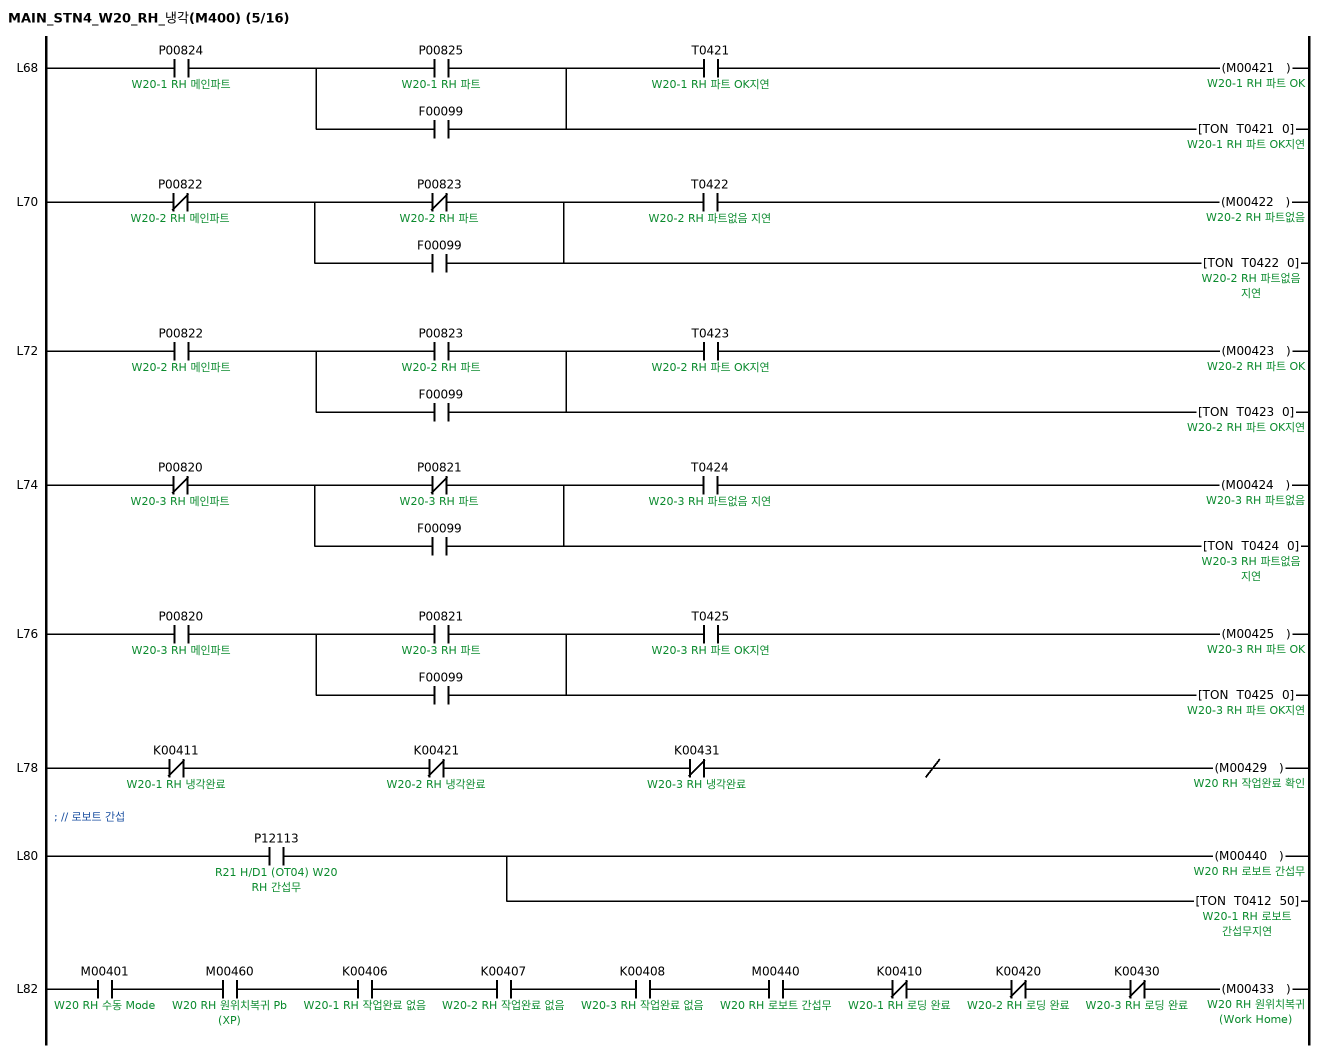
[picture p96: MAIN_STN4_W20_RH_냉각(M400) rungs L68-L82]
; L68
LOAD      P00824	// W20-1 RH 메인파트
LOAD      P00825	// W20-1 RH 파트
OR        F00099
AND LOAD
MPUSH
AND       T0421	// W20-1 RH 파트 OK지연
OUT       M00421	// W20-1 RH 파트 OK
MPOP
TON       T0421 0	// W20-1 RH 파트 OK지연
; L70
LOAD NOT  P00822	// W20-2 RH 메인파트
LOAD NOT  P00823	// W20-2 RH 파트
OR        F00099
AND LOAD
MPUSH
AND       T0422	// W20-2 RH 파트없음 지연
OUT       M00422	// W20-2 RH 파트없음
MPOP
TON       T0422 0	// W20-2 RH 파트없음 지연
; L72
LOAD      P00822	// W20-2 RH 메인파트
LOAD      P00823	// W20-2 RH 파트
OR        F00099
AND LOAD
MPUSH
AND       T0423	// W20-2 RH 파트 OK지연
OUT       M00423	// W20-2 RH 파트 OK
MPOP
TON       T0423 0	// W20-2 RH 파트 OK지연
; L74
LOAD NOT  P00820	// W20-3 RH 메인파트
LOAD NOT  P00821	// W20-3 RH 파트
OR        F00099
AND LOAD
MPUSH
AND       T0424	// W20-3 RH 파트없음 지연
OUT       M00424	// W20-3 RH 파트없음
MPOP
TON       T0424 0	// W20-3 RH 파트없음 지연
; L76
LOAD      P00820	// W20-3 RH 메인파트
LOAD      P00821	// W20-3 RH 파트
OR        F00099
AND LOAD
MPUSH
AND       T0425	// W20-3 RH 파트 OK지연
OUT       M00425	// W20-3 RH 파트 OK
MPOP
TON       T0425 0	// W20-3 RH 파트 OK지연
; L78
LOAD NOT  K00411	// W20-1 RH 냉각완료
AND NOT   K00421	// W20-2 RH 냉각완료
AND NOT   K00431	// W20-3 RH 냉각완료
NOT
OUT       M00429	// W20 RH 작업완료 확인
//   // 로보트 간섭
; L80
LOAD      P12113	// R21 H/D1 (OT04) W20 RH 간섭무
OUT       M00440	// W20 RH 로보트 간섭무
TON       T0412 50	// W20-1 RH 로보트 간섭무지연
; L82
LOAD      M00401	// W20 RH 수동 Mode
AND       M00460	// W20 RH 원위치복귀 Pb (XP)
AND       K00406	// W20-1 RH 작업완료 없음
AND       K00407	// W20-2 RH 작업완료 없음
AND       K00408	// W20-3 RH 작업완료 없음
AND       M00440	// W20 RH 로보트 간섭무
AND NOT   K00410	// W20-1 RH 로딩 완료
AND NOT   K00420	// W20-2 RH 로딩 완료
AND NOT   K00430	// W20-3 RH 로딩 완료
OUT       M00433	// W20 RH 원위치복귀 (Work Home)

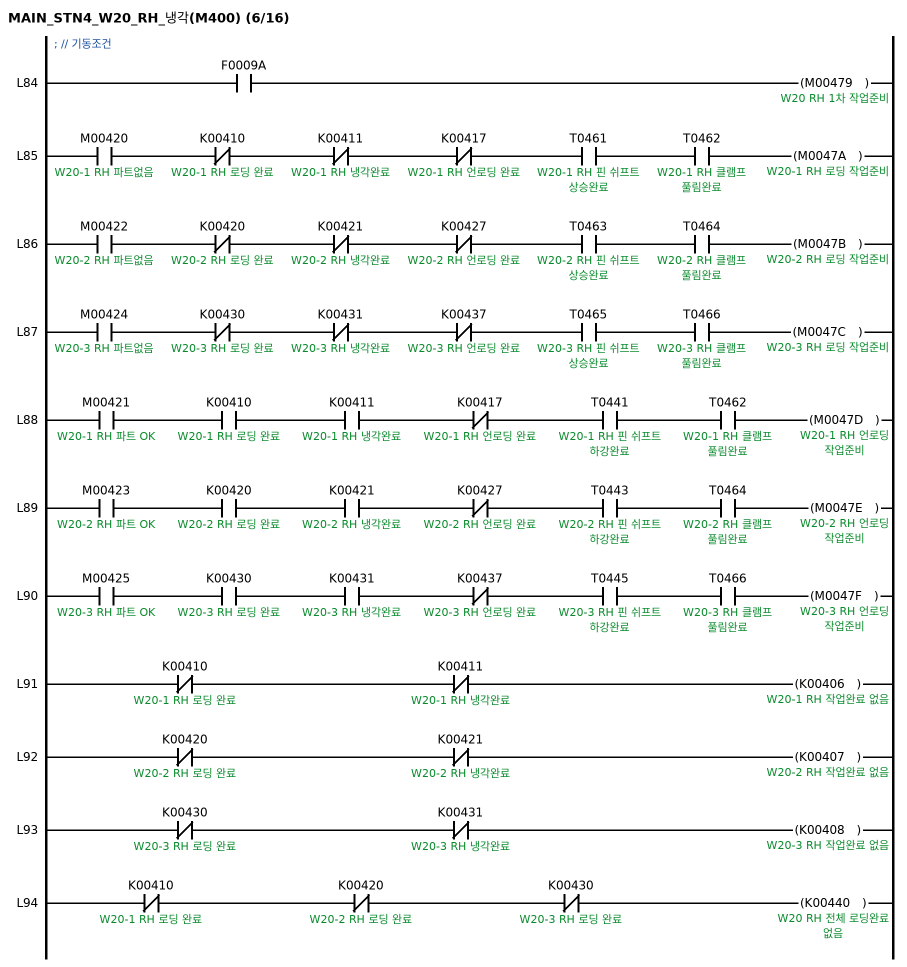
//   // 기동조건
; L84
LOAD      F0009A
OUT       M00479	// W20 RH 1차 작업준비
; L85
LOAD      M00420	// W20-1 RH 파트없음
AND NOT   K00410	// W20-1 RH 로딩 완료
AND NOT   K00411	// W20-1 RH 냉각완료
AND NOT   K00417	// W20-1 RH 언로딩 완료
AND       T0461	// W20-1 RH 핀 쉬프트 상승완료
AND       T0462	// W20-1 RH 클램프 풀림완료
OUT       M0047A	// W20-1 RH 로딩 작업준비
; L86
LOAD      M00422	// W20-2 RH 파트없음
AND NOT   K00420	// W20-2 RH 로딩 완료
AND NOT   K00421	// W20-2 RH 냉각완료
AND NOT   K00427	// W20-2 RH 언로딩 완료
AND       T0463	// W20-2 RH 핀 쉬프트 상승완료
AND       T0464	// W20-2 RH 클램프 풀림완료
OUT       M0047B	// W20-2 RH 로딩 작업준비
; L87
LOAD      M00424	// W20-3 RH 파트없음
AND NOT   K00430	// W20-3 RH 로딩 완료
AND NOT   K00431	// W20-3 RH 냉각완료
AND NOT   K00437	// W20-3 RH 언로딩 완료
AND       T0465	// W20-3 RH 핀 쉬프트 상승완료
AND       T0466	// W20-3 RH 클램프 풀림완료
OUT       M0047C	// W20-3 RH 로딩 작업준비
; L88
LOAD      M00421	// W20-1 RH 파트 OK
AND       K00410	// W20-1 RH 로딩 완료
AND       K00411	// W20-1 RH 냉각완료
AND NOT   K00417	// W20-1 RH 언로딩 완료
AND       T0441	// W20-1 RH 핀 쉬프트 하강완료
AND       T0462	// W20-1 RH 클램프 풀림완료
OUT       M0047D	// W20-1 RH 언로딩 작업준비
; L89
LOAD      M00423	// W20-2 RH 파트 OK
AND       K00420	// W20-2 RH 로딩 완료
AND       K00421	// W20-2 RH 냉각완료
AND NOT   K00427	// W20-2 RH 언로딩 완료
AND       T0443	// W20-2 RH 핀 쉬프트 하강완료
AND       T0464	// W20-2 RH 클램프 풀림완료
OUT       M0047E	// W20-2 RH 언로딩 작업준비
; L90
LOAD      M00425	// W20-3 RH 파트 OK
AND       K00430	// W20-3 RH 로딩 완료
AND       K00431	// W20-3 RH 냉각완료
AND NOT   K00437	// W20-3 RH 언로딩 완료
AND       T0445	// W20-3 RH 핀 쉬프트 하강완료
AND       T0466	// W20-3 RH 클램프 풀림완료
OUT       M0047F	// W20-3 RH 언로딩 작업준비
; L91
LOAD NOT  K00410	// W20-1 RH 로딩 완료
AND NOT   K00411	// W20-1 RH 냉각완료
OUT       K00406	// W20-1 RH 작업완료 없음
; L92
LOAD NOT  K00420	// W20-2 RH 로딩 완료
AND NOT   K00421	// W20-2 RH 냉각완료
OUT       K00407	// W20-2 RH 작업완료 없음
; L93
LOAD NOT  K00430	// W20-3 RH 로딩 완료
AND NOT   K00431	// W20-3 RH 냉각완료
OUT       K00408	// W20-3 RH 작업완료 없음
; L94
LOAD NOT  K00410	// W20-1 RH 로딩 완료
AND NOT   K00420	// W20-2 RH 로딩 완료
AND NOT   K00430	// W20-3 RH 로딩 완료
OUT       K00440	// W20 RH 전체 로딩완료 없음

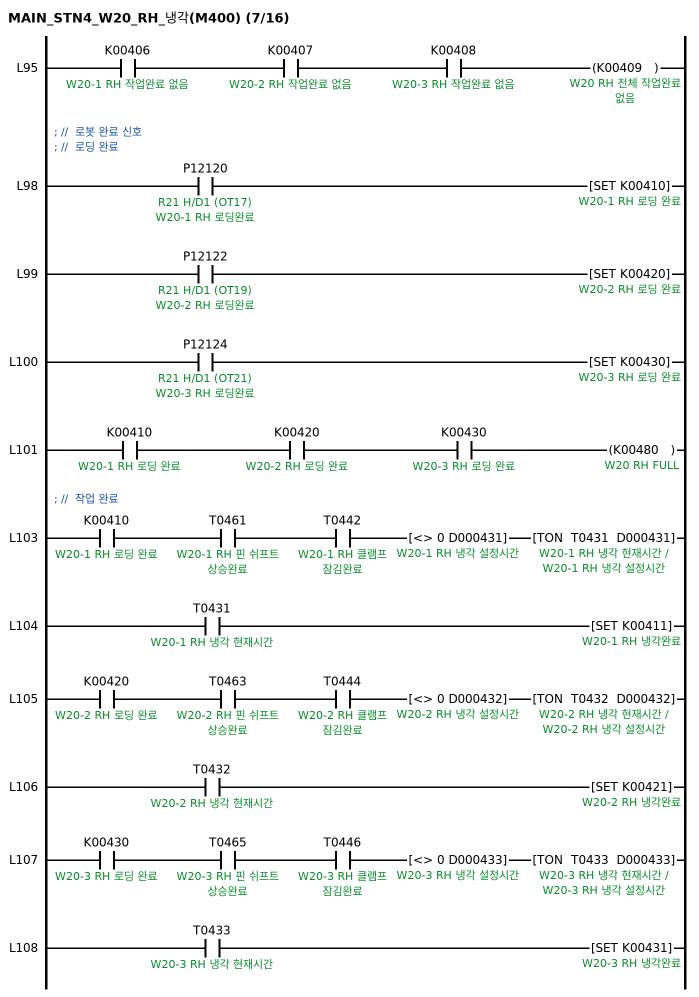
; L95
LOAD      K00406	// W20-1 RH 작업완료 없음
AND       K00407	// W20-2 RH 작업완료 없음
AND       K00408	// W20-3 RH 작업완료 없음
OUT       K00409	// W20 RH 전체 작업완료 없음
//   //  로봇 완료 신호
//   //  로딩 완료
; L98
LOAD      P12120	// R21 H/D1 (OT17) W20-1 RH 로딩완료
SET       K00410	// W20-1 RH 로딩 완료
; L99
LOAD      P12122	// R21 H/D1 (OT19) W20-2 RH 로딩완료
SET       K00420	// W20-2 RH 로딩 완료
; L100
LOAD      P12124	// R21 H/D1 (OT21) W20-3 RH 로딩완료
SET       K00430	// W20-3 RH 로딩 완료
; L101
LOAD      K00410	// W20-1 RH 로딩 완료
AND       K00420	// W20-2 RH 로딩 완료
AND       K00430	// W20-3 RH 로딩 완료
OUT       K00480	// W20 RH FULL
//   //  작업 완료
; L103
LOAD      K00410	// W20-1 RH 로딩 완료
AND       T0461	// W20-1 RH 핀 쉬프트 상승완료
AND       T0442	// W20-1 RH 클램프 잠김완료
AND<>     0 D000431	// W20-1 RH 냉각 설정시간
TON       T0431 D000431	// W20-1 RH 냉각 현재시간 / W20-1 RH 냉각 설정시간
; L104
LOAD      T0431	// W20-1 RH 냉각 현재시간
SET       K00411	// W20-1 RH 냉각완료
; L105
LOAD      K00420	// W20-2 RH 로딩 완료
AND       T0463	// W20-2 RH 핀 쉬프트 상승완료
AND       T0444	// W20-2 RH 클램프 잠김완료
AND<>     0 D000432	// W20-2 RH 냉각 설정시간
TON       T0432 D000432	// W20-2 RH 냉각 현재시간 / W20-2 RH 냉각 설정시간
; L106
LOAD      T0432	// W20-2 RH 냉각 현재시간
SET       K00421	// W20-2 RH 냉각완료
; L107
LOAD      K00430	// W20-3 RH 로딩 완료
AND       T0465	// W20-3 RH 핀 쉬프트 상승완료
AND       T0446	// W20-3 RH 클램프 잠김완료
AND<>     0 D000433	// W20-3 RH 냉각 설정시간
TON       T0433 D000433	// W20-3 RH 냉각 현재시간 / W20-3 RH 냉각 설정시간
; L108
LOAD      T0433	// W20-3 RH 냉각 현재시간
SET       K00431	// W20-3 RH 냉각완료

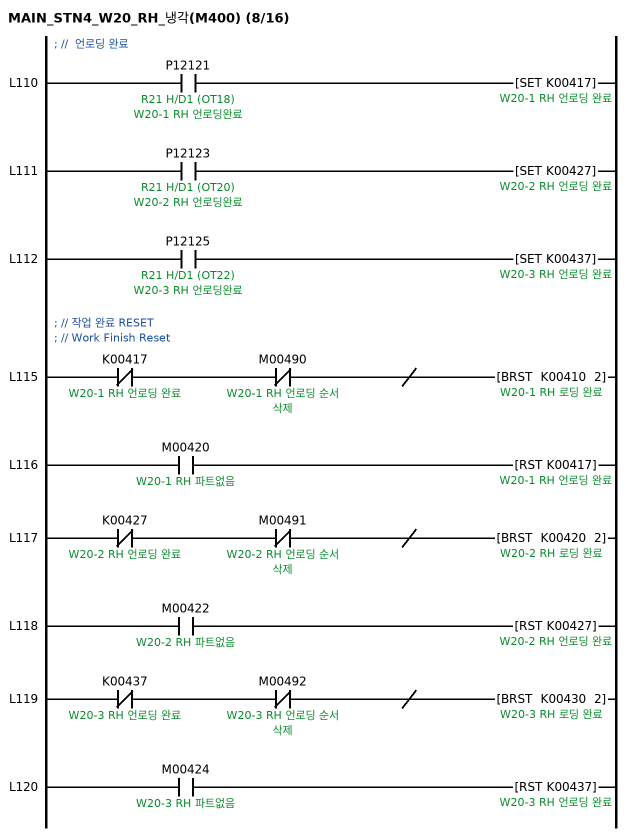
//   //  언로딩 완료
; L110
LOAD      P12121	// R21 H/D1 (OT18) W20-1 RH 언로딩완료
SET       K00417	// W20-1 RH 언로딩 완료
; L111
LOAD      P12123	// R21 H/D1 (OT20) W20-2 RH 언로딩완료
SET       K00427	// W20-2 RH 언로딩 완료
; L112
LOAD      P12125	// R21 H/D1 (OT22) W20-3 RH 언로딩완료
SET       K00437	// W20-3 RH 언로딩 완료
//     // 작업 완료 RESET
//   // Work Finish Reset
; L115
LOAD NOT  K00417	// W20-1 RH 언로딩 완료
AND NOT   M00490	// W20-1 RH 언로딩 순서 삭제
NOT
BRST      K00410 2	// W20-1 RH 로딩 완료
; L116
LOAD      M00420	// W20-1 RH 파트없음
RST       K00417	// W20-1 RH 언로딩 완료
; L117
LOAD NOT  K00427	// W20-2 RH 언로딩 완료
AND NOT   M00491	// W20-2 RH 언로딩 순서 삭제
NOT
BRST      K00420 2	// W20-2 RH 로딩 완료
; L118
LOAD      M00422	// W20-2 RH 파트없음
RST       K00427	// W20-2 RH 언로딩 완료
; L119
LOAD NOT  K00437	// W20-3 RH 언로딩 완료
AND NOT   M00492	// W20-3 RH 언로딩 순서 삭제
NOT
BRST      K00430 2	// W20-3 RH 로딩 완료
; L120
LOAD      M00424	// W20-3 RH 파트없음
RST       K00437	// W20-3 RH 언로딩 완료

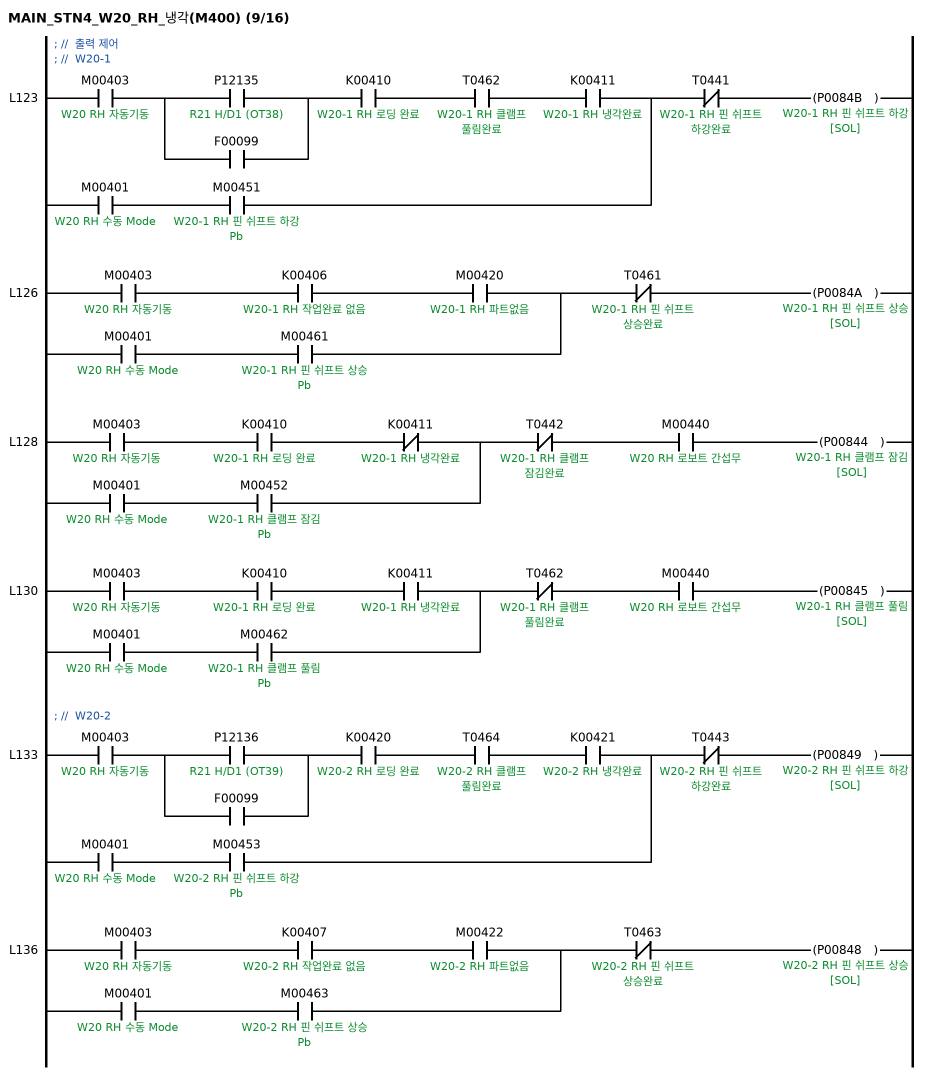
//     //  출력 제어
//     //  W20-1
; L123
LOAD      M00403	// W20 RH 자동기동
LOAD      P12135	// R21 H/D1 (OT38)
OR        F00099
AND LOAD
AND       K00410	// W20-1 RH 로딩 완료
AND       T0462	// W20-1 RH 클램프 풀림완료
AND       K00411	// W20-1 RH 냉각완료
LOAD      M00401	// W20 RH 수동 Mode
AND       M00451	// W20-1 RH 핀 쉬프트 하강 Pb
OR LOAD
AND NOT   T0441	// W20-1 RH 핀 쉬프트 하강완료
OUT       P0084B	// W20-1 RH 핀 쉬프트 하강 [SOL]
; L126
LOAD      M00403	// W20 RH 자동기동
AND       K00406	// W20-1 RH 작업완료 없음
AND       M00420	// W20-1 RH 파트없음
LOAD      M00401	// W20 RH 수동 Mode
AND       M00461	// W20-1 RH 핀 쉬프트 상승 Pb
OR LOAD
AND NOT   T0461	// W20-1 RH 핀 쉬프트 상승완료
OUT       P0084A	// W20-1 RH 핀 쉬프트 상승 [SOL]
; L128
LOAD      M00403	// W20 RH 자동기동
AND       K00410	// W20-1 RH 로딩 완료
AND NOT   K00411	// W20-1 RH 냉각완료
LOAD      M00401	// W20 RH 수동 Mode
AND       M00452	// W20-1 RH 클램프 잠김 Pb
OR LOAD
AND NOT   T0442	// W20-1 RH 클램프 잠김완료
AND       M00440	// W20 RH 로보트 간섭무
OUT       P00844	// W20-1 RH 클램프 잠김 [SOL]
; L130
LOAD      M00403	// W20 RH 자동기동
AND       K00410	// W20-1 RH 로딩 완료
AND       K00411	// W20-1 RH 냉각완료
LOAD      M00401	// W20 RH 수동 Mode
AND       M00462	// W20-1 RH 클램프 풀림 Pb
OR LOAD
AND NOT   T0462	// W20-1 RH 클램프 풀림완료
AND       M00440	// W20 RH 로보트 간섭무
OUT       P00845	// W20-1 RH 클램프 풀림 [SOL]
//     //  W20-2
; L133
LOAD      M00403	// W20 RH 자동기동
LOAD      P12136	// R21 H/D1 (OT39)
OR        F00099
AND LOAD
AND       K00420	// W20-2 RH 로딩 완료
AND       T0464	// W20-2 RH 클램프 풀림완료
AND       K00421	// W20-2 RH 냉각완료
LOAD      M00401	// W20 RH 수동 Mode
AND       M00453	// W20-2 RH 핀 쉬프트 하강 Pb
OR LOAD
AND NOT   T0443	// W20-2 RH 핀 쉬프트 하강완료
OUT       P00849	// W20-2 RH 핀 쉬프트 하강 [SOL]
; L136
LOAD      M00403	// W20 RH 자동기동
AND       K00407	// W20-2 RH 작업완료 없음
AND       M00422	// W20-2 RH 파트없음
LOAD      M00401	// W20 RH 수동 Mode
AND       M00463	// W20-2 RH 핀 쉬프트 상승 Pb
OR LOAD
AND NOT   T0463	// W20-2 RH 핀 쉬프트 상승완료
OUT       P00848	// W20-2 RH 핀 쉬프트 상승 [SOL]

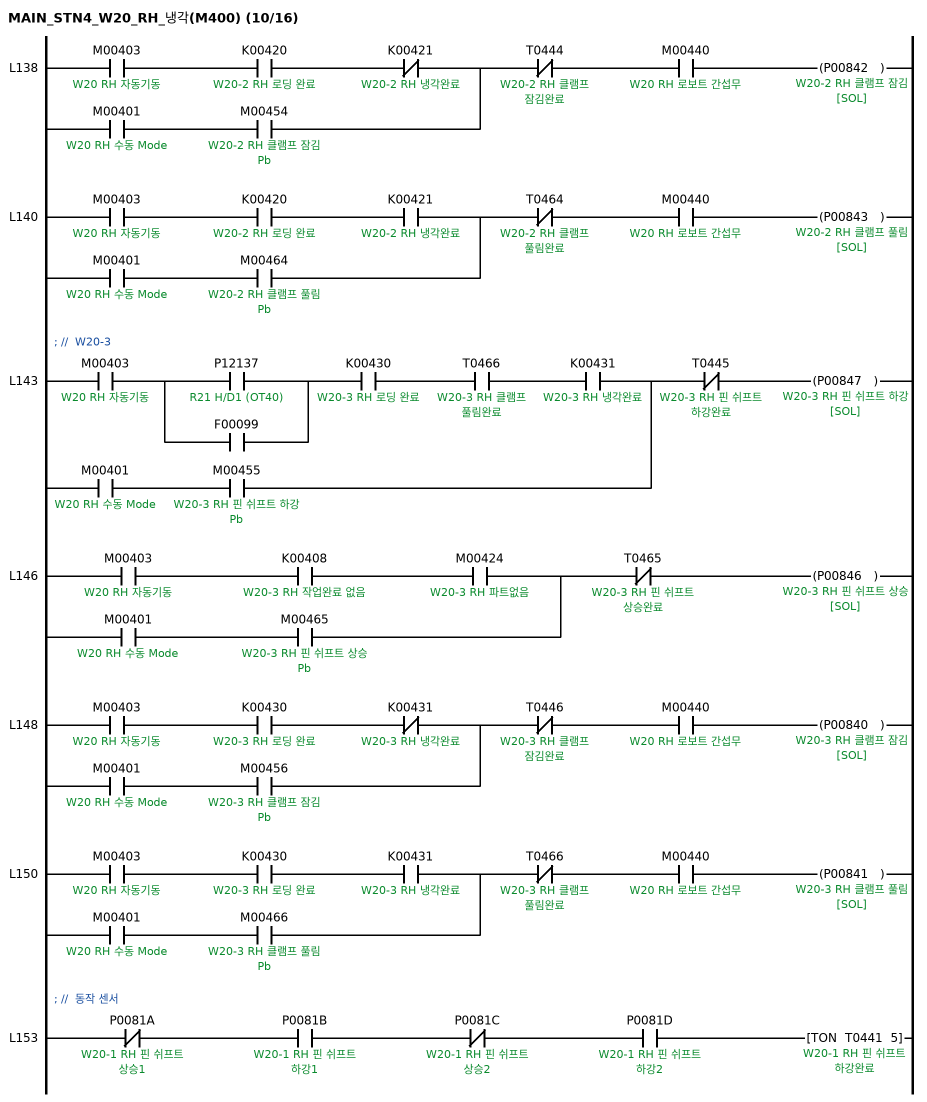
; L138
LOAD      M00403	// W20 RH 자동기동
AND       K00420	// W20-2 RH 로딩 완료
AND NOT   K00421	// W20-2 RH 냉각완료
LOAD      M00401	// W20 RH 수동 Mode
AND       M00454	// W20-2 RH 클램프 잠김 Pb
OR LOAD
AND NOT   T0444	// W20-2 RH 클램프 잠김완료
AND       M00440	// W20 RH 로보트 간섭무
OUT       P00842	// W20-2 RH 클램프 잠김 [SOL]
; L140
LOAD      M00403	// W20 RH 자동기동
AND       K00420	// W20-2 RH 로딩 완료
AND       K00421	// W20-2 RH 냉각완료
LOAD      M00401	// W20 RH 수동 Mode
AND       M00464	// W20-2 RH 클램프 풀림 Pb
OR LOAD
AND NOT   T0464	// W20-2 RH 클램프 풀림완료
AND       M00440	// W20 RH 로보트 간섭무
OUT       P00843	// W20-2 RH 클램프 풀림 [SOL]
//     //  W20-3
; L143
LOAD      M00403	// W20 RH 자동기동
LOAD      P12137	// R21 H/D1 (OT40)
OR        F00099
AND LOAD
AND       K00430	// W20-3 RH 로딩 완료
AND       T0466	// W20-3 RH 클램프 풀림완료
AND       K00431	// W20-3 RH 냉각완료
LOAD      M00401	// W20 RH 수동 Mode
AND       M00455	// W20-3 RH 핀 쉬프트 하강 Pb
OR LOAD
AND NOT   T0445	// W20-3 RH 핀 쉬프트 하강완료
OUT       P00847	// W20-3 RH 핀 쉬프트 하강 [SOL]
; L146
LOAD      M00403	// W20 RH 자동기동
AND       K00408	// W20-3 RH 작업완료 없음
AND       M00424	// W20-3 RH 파트없음
LOAD      M00401	// W20 RH 수동 Mode
AND       M00465	// W20-3 RH 핀 쉬프트 상승 Pb
OR LOAD
AND NOT   T0465	// W20-3 RH 핀 쉬프트 상승완료
OUT       P00846	// W20-3 RH 핀 쉬프트 상승 [SOL]
; L148
LOAD      M00403	// W20 RH 자동기동
AND       K00430	// W20-3 RH 로딩 완료
AND NOT   K00431	// W20-3 RH 냉각완료
LOAD      M00401	// W20 RH 수동 Mode
AND       M00456	// W20-3 RH 클램프 잠김 Pb
OR LOAD
AND NOT   T0446	// W20-3 RH 클램프 잠김완료
AND       M00440	// W20 RH 로보트 간섭무
OUT       P00840	// W20-3 RH 클램프 잠김 [SOL]
; L150
LOAD      M00403	// W20 RH 자동기동
AND       K00430	// W20-3 RH 로딩 완료
AND       K00431	// W20-3 RH 냉각완료
LOAD      M00401	// W20 RH 수동 Mode
AND       M00466	// W20-3 RH 클램프 풀림 Pb
OR LOAD
AND NOT   T0466	// W20-3 RH 클램프 풀림완료
AND       M00440	// W20 RH 로보트 간섭무
OUT       P00841	// W20-3 RH 클램프 풀림 [SOL]
//   //  동작 센서
; L153
LOAD NOT  P0081A	// W20-1 RH 핀 쉬프트 상승1
AND       P0081B	// W20-1 RH 핀 쉬프트 하강1
AND NOT   P0081C	// W20-1 RH 핀 쉬프트 상승2
AND       P0081D	// W20-1 RH 핀 쉬프트 하강2
TON       T0441 5	// W20-1 RH 핀 쉬프트 하강완료

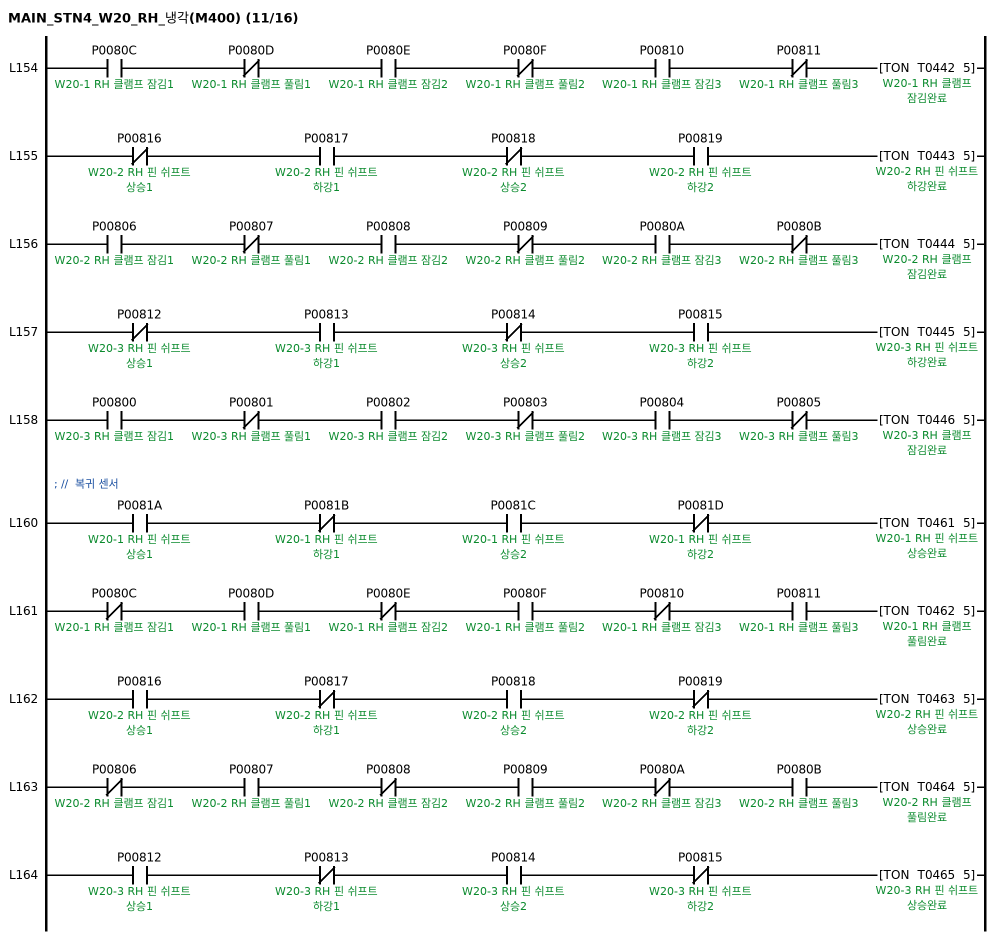
; L154
LOAD      P0080C	// W20-1 RH 클램프 잠김1
AND NOT   P0080D	// W20-1 RH 클램프 풀림1
AND       P0080E	// W20-1 RH 클램프 잠김2
AND NOT   P0080F	// W20-1 RH 클램프 풀림2
AND       P00810	// W20-1 RH 클램프 잠김3
AND NOT   P00811	// W20-1 RH 클램프 풀림3
TON       T0442 5	// W20-1 RH 클램프 잠김완료
; L155
LOAD NOT  P00816	// W20-2 RH 핀 쉬프트 상승1
AND       P00817	// W20-2 RH 핀 쉬프트 하강1
AND NOT   P00818	// W20-2 RH 핀 쉬프트 상승2
AND       P00819	// W20-2 RH 핀 쉬프트 하강2
TON       T0443 5	// W20-2 RH 핀 쉬프트 하강완료
; L156
LOAD      P00806	// W20-2 RH 클램프 잠김1
AND NOT   P00807	// W20-2 RH 클램프 풀림1
AND       P00808	// W20-2 RH 클램프 잠김2
AND NOT   P00809	// W20-2 RH 클램프 풀림2
AND       P0080A	// W20-2 RH 클램프 잠김3
AND NOT   P0080B	// W20-2 RH 클램프 풀림3
TON       T0444 5	// W20-2 RH 클램프 잠김완료
; L157
LOAD NOT  P00812	// W20-3 RH 핀 쉬프트 상승1
AND       P00813	// W20-3 RH 핀 쉬프트 하강1
AND NOT   P00814	// W20-3 RH 핀 쉬프트 상승2
AND       P00815	// W20-3 RH 핀 쉬프트 하강2
TON       T0445 5	// W20-3 RH 핀 쉬프트 하강완료
; L158
LOAD      P00800	// W20-3 RH 클램프 잠김1
AND NOT   P00801	// W20-3 RH 클램프 풀림1
AND       P00802	// W20-3 RH 클램프 잠김2
AND NOT   P00803	// W20-3 RH 클램프 풀림2
AND       P00804	// W20-3 RH 클램프 잠김3
AND NOT   P00805	// W20-3 RH 클램프 풀림3
TON       T0446 5	// W20-3 RH 클램프 잠김완료
//   //  복귀 센서
; L160
LOAD      P0081A	// W20-1 RH 핀 쉬프트 상승1
AND NOT   P0081B	// W20-1 RH 핀 쉬프트 하강1
AND       P0081C	// W20-1 RH 핀 쉬프트 상승2
AND NOT   P0081D	// W20-1 RH 핀 쉬프트 하강2
TON       T0461 5	// W20-1 RH 핀 쉬프트 상승완료
; L161
LOAD NOT  P0080C	// W20-1 RH 클램프 잠김1
AND       P0080D	// W20-1 RH 클램프 풀림1
AND NOT   P0080E	// W20-1 RH 클램프 잠김2
AND       P0080F	// W20-1 RH 클램프 풀림2
AND NOT   P00810	// W20-1 RH 클램프 잠김3
AND       P00811	// W20-1 RH 클램프 풀림3
TON       T0462 5	// W20-1 RH 클램프 풀림완료
; L162
LOAD      P00816	// W20-2 RH 핀 쉬프트 상승1
AND NOT   P00817	// W20-2 RH 핀 쉬프트 하강1
AND       P00818	// W20-2 RH 핀 쉬프트 상승2
AND NOT   P00819	// W20-2 RH 핀 쉬프트 하강2
TON       T0463 5	// W20-2 RH 핀 쉬프트 상승완료
; L163
LOAD NOT  P00806	// W20-2 RH 클램프 잠김1
AND       P00807	// W20-2 RH 클램프 풀림1
AND NOT   P00808	// W20-2 RH 클램프 잠김2
AND       P00809	// W20-2 RH 클램프 풀림2
AND NOT   P0080A	// W20-2 RH 클램프 잠김3
AND       P0080B	// W20-2 RH 클램프 풀림3
TON       T0464 5	// W20-2 RH 클램프 풀림완료
; L164
LOAD      P00812	// W20-3 RH 핀 쉬프트 상승1
AND NOT   P00813	// W20-3 RH 핀 쉬프트 하강1
AND       P00814	// W20-3 RH 핀 쉬프트 상승2
AND NOT   P00815	// W20-3 RH 핀 쉬프트 하강2
TON       T0465 5	// W20-3 RH 핀 쉬프트 상승완료

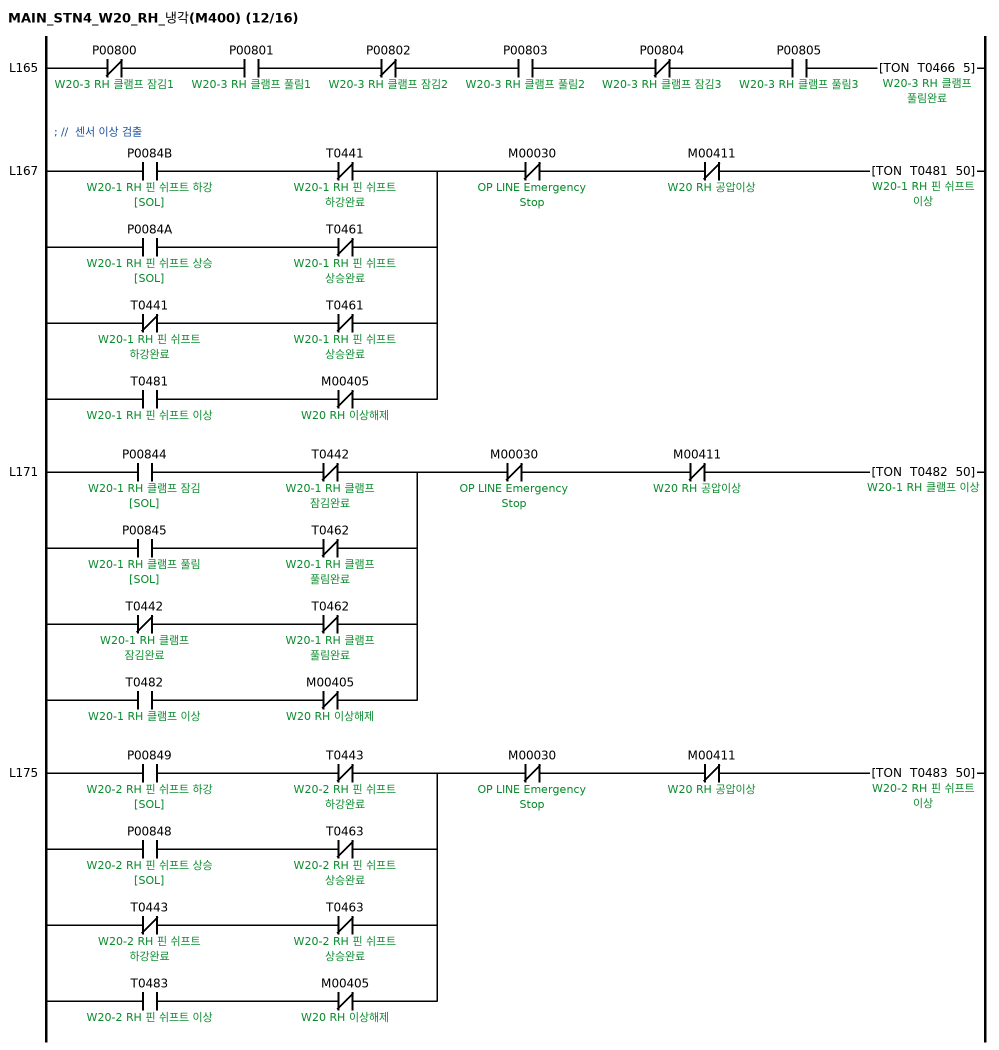
; L165
LOAD NOT  P00800	// W20-3 RH 클램프 잠김1
AND       P00801	// W20-3 RH 클램프 풀림1
AND NOT   P00802	// W20-3 RH 클램프 잠김2
AND       P00803	// W20-3 RH 클램프 풀림2
AND NOT   P00804	// W20-3 RH 클램프 잠김3
AND       P00805	// W20-3 RH 클램프 풀림3
TON       T0466 5	// W20-3 RH 클램프 풀림완료
//     //  센서 이상 검출
; L167
LOAD      P0084B	// W20-1 RH 핀 쉬프트 하강 [SOL]
AND NOT   T0441	// W20-1 RH 핀 쉬프트 하강완료
LOAD      P0084A	// W20-1 RH 핀 쉬프트 상승 [SOL]
AND NOT   T0461	// W20-1 RH 핀 쉬프트 상승완료
OR LOAD
LOAD NOT  T0441	// W20-1 RH 핀 쉬프트 하강완료
AND NOT   T0461	// W20-1 RH 핀 쉬프트 상승완료
OR LOAD
LOAD      T0481	// W20-1 RH 핀 쉬프트 이상
AND NOT   M00405	// W20 RH 이상해제
OR LOAD
AND NOT   M00030	// OP LINE Emergency Stop
AND NOT   M00411	// W20 RH 공압이상
TON       T0481 50	// W20-1 RH 핀 쉬프트 이상
; L171
LOAD      P00844	// W20-1 RH 클램프 잠김 [SOL]
AND NOT   T0442	// W20-1 RH 클램프 잠김완료
LOAD      P00845	// W20-1 RH 클램프 풀림 [SOL]
AND NOT   T0462	// W20-1 RH 클램프 풀림완료
OR LOAD
LOAD NOT  T0442	// W20-1 RH 클램프 잠김완료
AND NOT   T0462	// W20-1 RH 클램프 풀림완료
OR LOAD
LOAD      T0482	// W20-1 RH 클램프 이상
AND NOT   M00405	// W20 RH 이상해제
OR LOAD
AND NOT   M00030	// OP LINE Emergency Stop
AND NOT   M00411	// W20 RH 공압이상
TON       T0482 50	// W20-1 RH 클램프 이상
; L175
LOAD      P00849	// W20-2 RH 핀 쉬프트 하강 [SOL]
AND NOT   T0443	// W20-2 RH 핀 쉬프트 하강완료
LOAD      P00848	// W20-2 RH 핀 쉬프트 상승 [SOL]
AND NOT   T0463	// W20-2 RH 핀 쉬프트 상승완료
OR LOAD
LOAD NOT  T0443	// W20-2 RH 핀 쉬프트 하강완료
AND NOT   T0463	// W20-2 RH 핀 쉬프트 상승완료
OR LOAD
LOAD      T0483	// W20-2 RH 핀 쉬프트 이상
AND NOT   M00405	// W20 RH 이상해제
OR LOAD
AND NOT   M00030	// OP LINE Emergency Stop
AND NOT   M00411	// W20 RH 공압이상
TON       T0483 50	// W20-2 RH 핀 쉬프트 이상

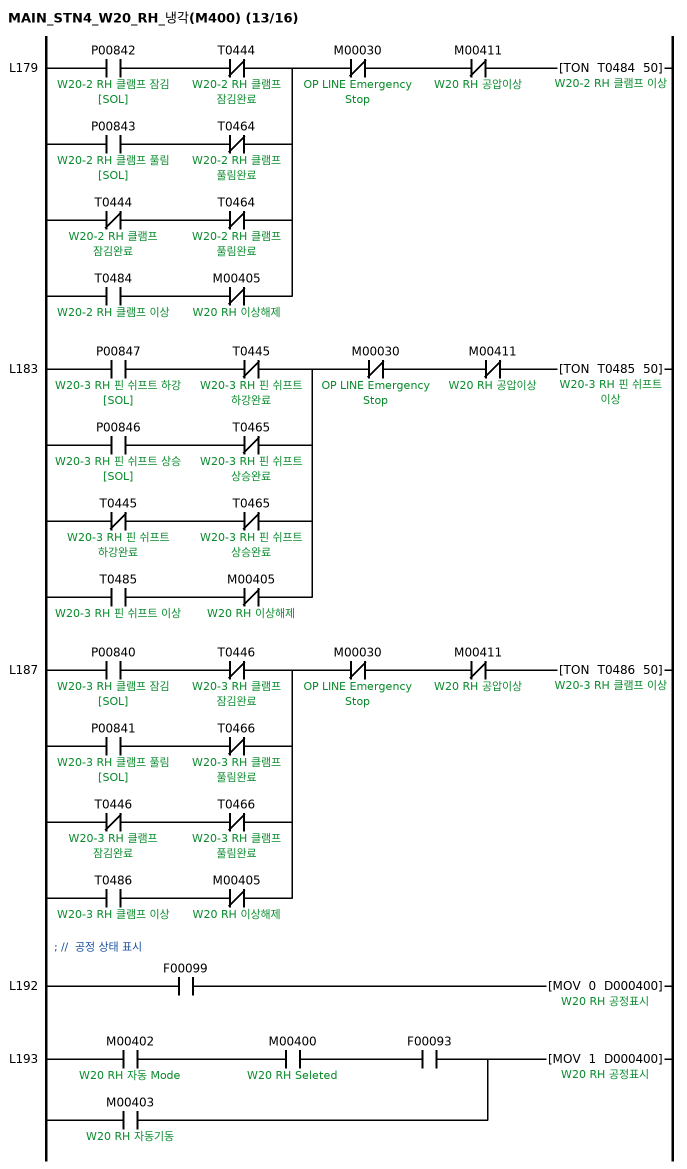
; L179
LOAD      P00842	// W20-2 RH 클램프 잠김 [SOL]
AND NOT   T0444	// W20-2 RH 클램프 잠김완료
LOAD      P00843	// W20-2 RH 클램프 풀림 [SOL]
AND NOT   T0464	// W20-2 RH 클램프 풀림완료
OR LOAD
LOAD NOT  T0444	// W20-2 RH 클램프 잠김완료
AND NOT   T0464	// W20-2 RH 클램프 풀림완료
OR LOAD
LOAD      T0484	// W20-2 RH 클램프 이상
AND NOT   M00405	// W20 RH 이상해제
OR LOAD
AND NOT   M00030	// OP LINE Emergency Stop
AND NOT   M00411	// W20 RH 공압이상
TON       T0484 50	// W20-2 RH 클램프 이상
; L183
LOAD      P00847	// W20-3 RH 핀 쉬프트 하강 [SOL]
AND NOT   T0445	// W20-3 RH 핀 쉬프트 하강완료
LOAD      P00846	// W20-3 RH 핀 쉬프트 상승 [SOL]
AND NOT   T0465	// W20-3 RH 핀 쉬프트 상승완료
OR LOAD
LOAD NOT  T0445	// W20-3 RH 핀 쉬프트 하강완료
AND NOT   T0465	// W20-3 RH 핀 쉬프트 상승완료
OR LOAD
LOAD      T0485	// W20-3 RH 핀 쉬프트 이상
AND NOT   M00405	// W20 RH 이상해제
OR LOAD
AND NOT   M00030	// OP LINE Emergency Stop
AND NOT   M00411	// W20 RH 공압이상
TON       T0485 50	// W20-3 RH 핀 쉬프트 이상
; L187
LOAD      P00840	// W20-3 RH 클램프 잠김 [SOL]
AND NOT   T0446	// W20-3 RH 클램프 잠김완료
LOAD      P00841	// W20-3 RH 클램프 풀림 [SOL]
AND NOT   T0466	// W20-3 RH 클램프 풀림완료
OR LOAD
LOAD NOT  T0446	// W20-3 RH 클램프 잠김완료
AND NOT   T0466	// W20-3 RH 클램프 풀림완료
OR LOAD
LOAD      T0486	// W20-3 RH 클램프 이상
AND NOT   M00405	// W20 RH 이상해제
OR LOAD
AND NOT   M00030	// OP LINE Emergency Stop
AND NOT   M00411	// W20 RH 공압이상
TON       T0486 50	// W20-3 RH 클램프 이상
//   //  공정 상태 표시
; L192
LOAD      F00099
MOV       0 D000400	// W20 RH 공정표시
; L193
LOAD      M00402	// W20 RH 자동 Mode
AND       M00400	// W20 RH Seleted
AND       F00093
OR        M00403	// W20 RH 자동기동
MOV       1 D000400	// W20 RH 공정표시

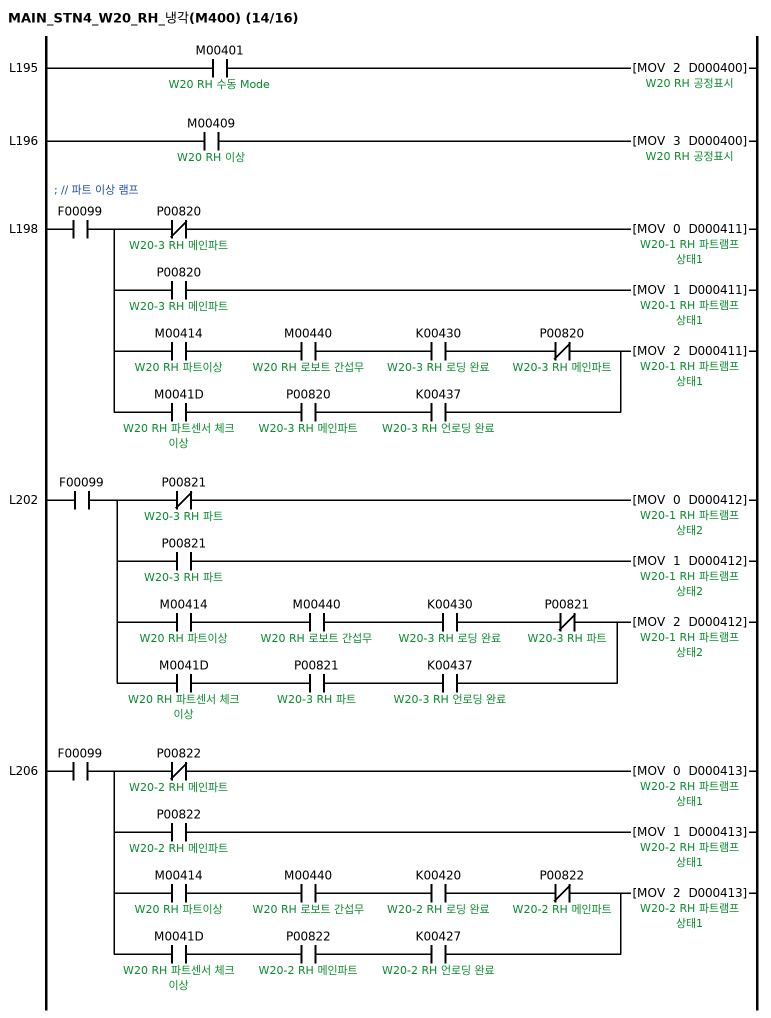
; L195
LOAD      M00401	// W20 RH 수동 Mode
MOV       2 D000400	// W20 RH 공정표시
; L196
LOAD      M00409	// W20 RH 이상
MOV       3 D000400	// W20 RH 공정표시
//   // 파트 이상 램프
; L198
LOAD      F00099
MPUSH
AND NOT   P00820	// W20-3 RH 메인파트
MOV       0 D000411	// W20-1 RH 파트램프 상태1
MLOAD
AND       P00820	// W20-3 RH 메인파트
MOV       1 D000411	// W20-1 RH 파트램프 상태1
MPOP
LOAD      M00414	// W20 RH 파트이상
AND       M00440	// W20 RH 로보트 간섭무
AND       K00430	// W20-3 RH 로딩 완료
AND NOT   P00820	// W20-3 RH 메인파트
LOAD      M0041D	// W20 RH 파트센서 체크 이상
AND       P00820	// W20-3 RH 메인파트
AND       K00437	// W20-3 RH 언로딩 완료
OR LOAD
AND LOAD
MOV       2 D000411	// W20-1 RH 파트램프 상태1
; L202
LOAD      F00099
MPUSH
AND NOT   P00821	// W20-3 RH 파트
MOV       0 D000412	// W20-1 RH 파트램프 상태2
MLOAD
AND       P00821	// W20-3 RH 파트
MOV       1 D000412	// W20-1 RH 파트램프 상태2
MPOP
LOAD      M00414	// W20 RH 파트이상
AND       M00440	// W20 RH 로보트 간섭무
AND       K00430	// W20-3 RH 로딩 완료
AND NOT   P00821	// W20-3 RH 파트
LOAD      M0041D	// W20 RH 파트센서 체크 이상
AND       P00821	// W20-3 RH 파트
AND       K00437	// W20-3 RH 언로딩 완료
OR LOAD
AND LOAD
MOV       2 D000412	// W20-1 RH 파트램프 상태2
; L206
LOAD      F00099
MPUSH
AND NOT   P00822	// W20-2 RH 메인파트
MOV       0 D000413	// W20-2 RH 파트램프 상태1
MLOAD
AND       P00822	// W20-2 RH 메인파트
MOV       1 D000413	// W20-2 RH 파트램프 상태1
MPOP
LOAD      M00414	// W20 RH 파트이상
AND       M00440	// W20 RH 로보트 간섭무
AND       K00420	// W20-2 RH 로딩 완료
AND NOT   P00822	// W20-2 RH 메인파트
LOAD      M0041D	// W20 RH 파트센서 체크 이상
AND       P00822	// W20-2 RH 메인파트
AND       K00427	// W20-2 RH 언로딩 완료
OR LOAD
AND LOAD
MOV       2 D000413	// W20-2 RH 파트램프 상태1

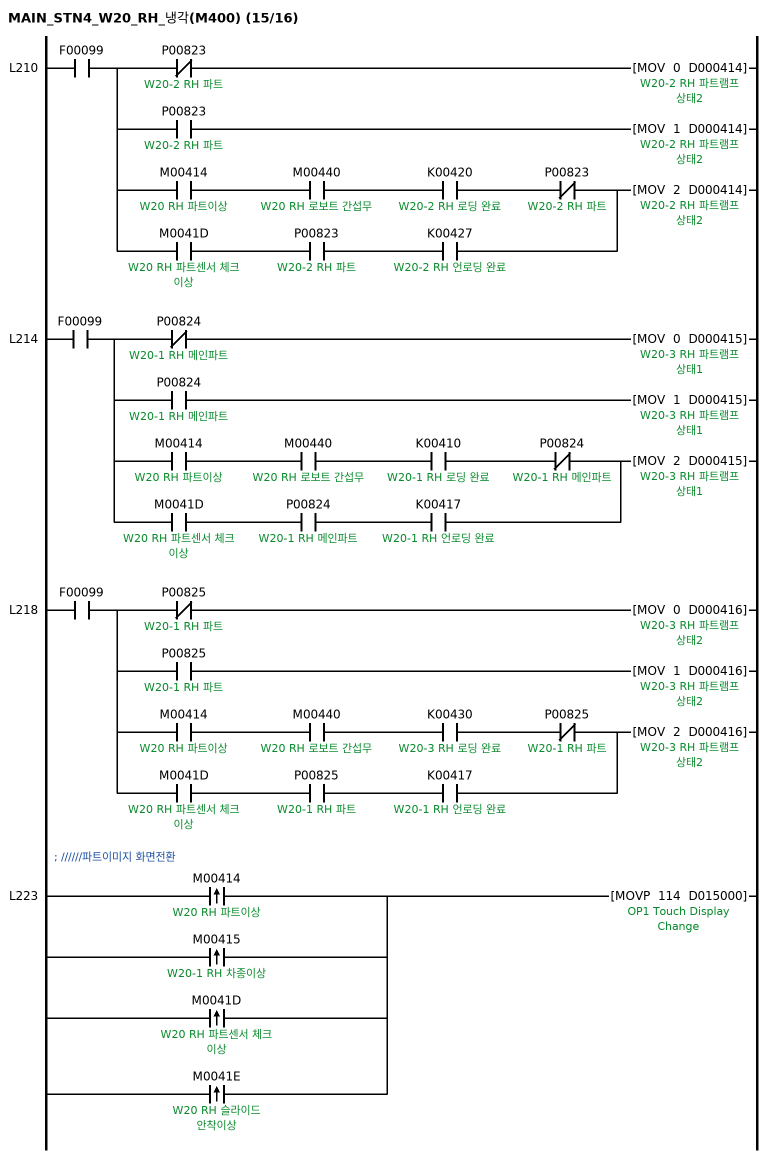
; L210
LOAD      F00099
MPUSH
AND NOT   P00823	// W20-2 RH 파트
MOV       0 D000414	// W20-2 RH 파트램프 상태2
MLOAD
AND       P00823	// W20-2 RH 파트
MOV       1 D000414	// W20-2 RH 파트램프 상태2
MPOP
LOAD      M00414	// W20 RH 파트이상
AND       M00440	// W20 RH 로보트 간섭무
AND       K00420	// W20-2 RH 로딩 완료
AND NOT   P00823	// W20-2 RH 파트
LOAD      M0041D	// W20 RH 파트센서 체크 이상
AND       P00823	// W20-2 RH 파트
AND       K00427	// W20-2 RH 언로딩 완료
OR LOAD
AND LOAD
MOV       2 D000414	// W20-2 RH 파트램프 상태2
; L214
LOAD      F00099
MPUSH
AND NOT   P00824	// W20-1 RH 메인파트
MOV       0 D000415	// W20-3 RH 파트램프 상태1
MLOAD
AND       P00824	// W20-1 RH 메인파트
MOV       1 D000415	// W20-3 RH 파트램프 상태1
MPOP
LOAD      M00414	// W20 RH 파트이상
AND       M00440	// W20 RH 로보트 간섭무
AND       K00410	// W20-1 RH 로딩 완료
AND NOT   P00824	// W20-1 RH 메인파트
LOAD      M0041D	// W20 RH 파트센서 체크 이상
AND       P00824	// W20-1 RH 메인파트
AND       K00417	// W20-1 RH 언로딩 완료
OR LOAD
AND LOAD
MOV       2 D000415	// W20-3 RH 파트램프 상태1
; L218
LOAD      F00099
MPUSH
AND NOT   P00825	// W20-1 RH 파트
MOV       0 D000416	// W20-3 RH 파트램프 상태2
MLOAD
AND       P00825	// W20-1 RH 파트
MOV       1 D000416	// W20-3 RH 파트램프 상태2
MPOP
LOAD      M00414	// W20 RH 파트이상
AND       M00440	// W20 RH 로보트 간섭무
AND       K00430	// W20-3 RH 로딩 완료
AND NOT   P00825	// W20-1 RH 파트
LOAD      M0041D	// W20 RH 파트센서 체크 이상
AND       P00825	// W20-1 RH 파트
AND       K00417	// W20-1 RH 언로딩 완료
OR LOAD
AND LOAD
MOV       2 D000416	// W20-3 RH 파트램프 상태2
// //////파트이미지 화면전환
; L223
LOADP     M00414	// W20 RH 파트이상
ORP       M00415	// W20-1 RH 차종이상
ORP       M0041D	// W20 RH 파트센서 체크 이상
ORP       M0041E	// W20 RH 슬라이드 안착이상
MOVP      114 D015000	// OP1 Touch Display Change

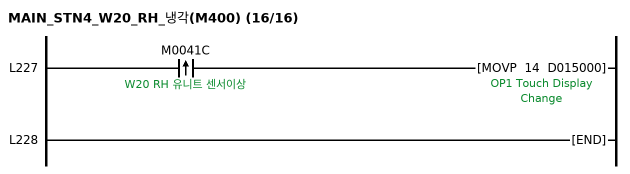
; L227
LOADP     M0041C	// W20 RH 유니트 센서이상
MOVP      14 D015000	// OP1 Touch Display Change
; L228
END

PROGRAM MAIN_STN5_W30_IDLE(M500) (task: 스캔 프로그램)

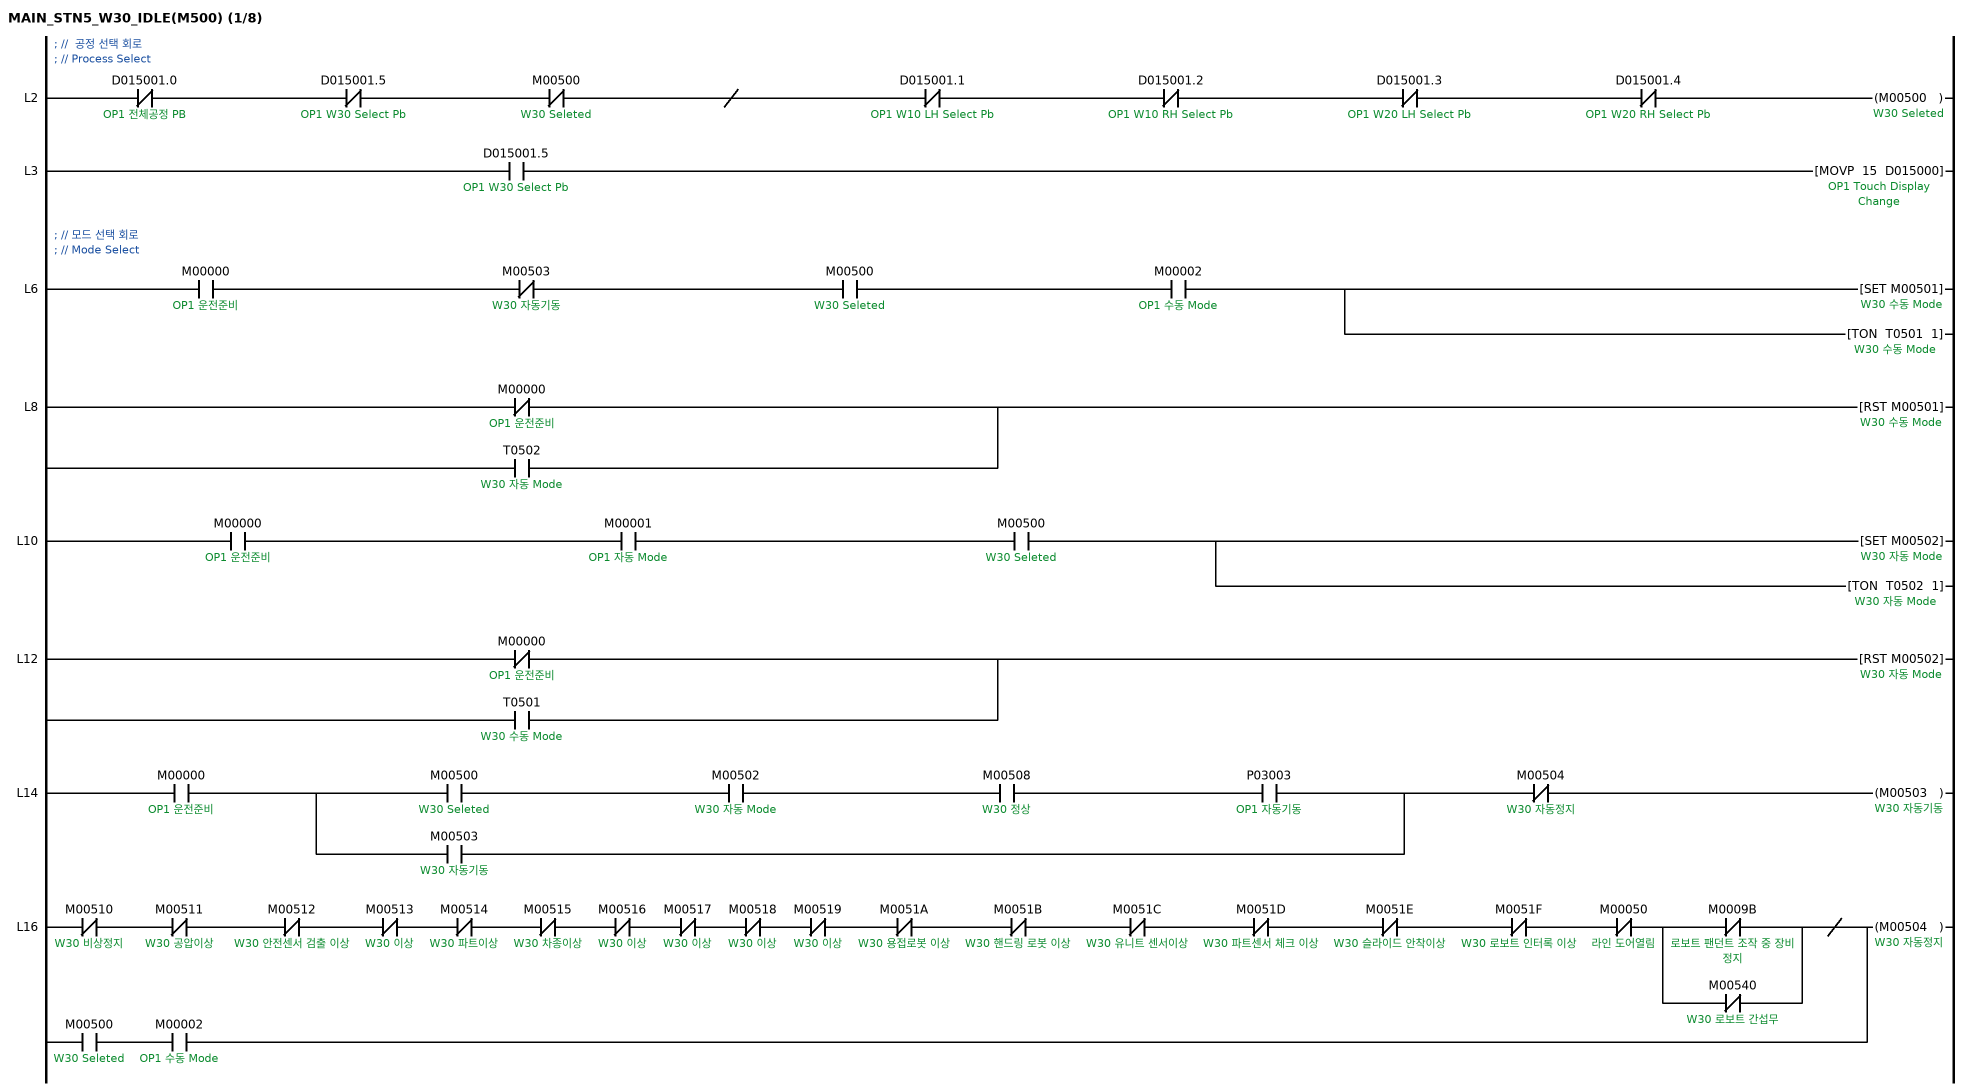
//   //  공정 선택 회로
//   // Process Select
; L2
LOAD NOT  D015001.0	// OP1 전체공정 PB
AND NOT   D015001.5	// OP1 W30 Select Pb
AND NOT   M00500	// W30 Seleted
NOT
AND NOT   D015001.1	// OP1 W10 LH Select Pb
AND NOT   D015001.2	// OP1 W10 RH Select Pb
AND NOT   D015001.3	// OP1 W20 LH Select Pb
AND NOT   D015001.4	// OP1 W20 RH Select Pb
OUT       M00500	// W30 Seleted
; L3
LOAD      D015001.5	// OP1 W30 Select Pb
MOVP      15 D015000	// OP1 Touch Display Change
// // 모드 선택 회로
//   // Mode Select
; L6
LOAD      M00000	// OP1 운전준비
AND NOT   M00503	// W30 자동기동
AND       M00500	// W30 Seleted
AND       M00002	// OP1 수동 Mode
SET       M00501	// W30 수동 Mode
TON       T0501 1	// W30 수동 Mode
; L8
LOAD NOT  M00000	// OP1 운전준비
OR        T0502	// W30 자동 Mode
RST       M00501	// W30 수동 Mode
; L10
LOAD      M00000	// OP1 운전준비
AND       M00001	// OP1 자동 Mode
AND       M00500	// W30 Seleted
SET       M00502	// W30 자동 Mode
TON       T0502 1	// W30 자동 Mode
; L12
LOAD NOT  M00000	// OP1 운전준비
OR        T0501	// W30 수동 Mode
RST       M00502	// W30 자동 Mode
; L14
LOAD      M00000	// OP1 운전준비
LOAD      M00500	// W30 Seleted
AND       M00502	// W30 자동 Mode
AND       M00508	// W30 정상
AND       P03003	// OP1 자동기동
OR        M00503	// W30 자동기동
AND LOAD
AND NOT   M00504	// W30 자동정지
OUT       M00503	// W30 자동기동
; L16
LOAD NOT  M00510	// W30 비상정지
AND NOT   M00511	// W30 공압이상
AND NOT   M00512	// W30 안전센서 검출 이상
AND NOT   M00513	// W30 이상
AND NOT   M00514	// W30 파트이상
AND NOT   M00515	// W30 차종이상
AND NOT   M00516	// W30 이상
AND NOT   M00517	// W30 이상
AND NOT   M00518	// W30 이상
AND NOT   M00519	// W30 이상
AND NOT   M0051A	// W30 용접로봇 이상
AND NOT   M0051B	// W30 핸드링 로봇 이상
AND NOT   M0051C	// W30 유니트 센서이상
AND NOT   M0051D	// W30 파트센서 체크 이상
AND NOT   M0051E	// W30 슬라이드 안착이상
AND NOT   M0051F	// W30 로보트 인터록 이상
AND NOT   M00050	// 라인 도어열림
LOAD NOT  M0009B	// 로보트 팬던트 조작 중 장비 정지
OR NOT    M00540	// W30 로보트 간섭무
AND LOAD
NOT
LOAD      M00500	// W30 Seleted
AND       M00002	// OP1 수동 Mode
OR LOAD
OUT       M00504	// W30 자동정지

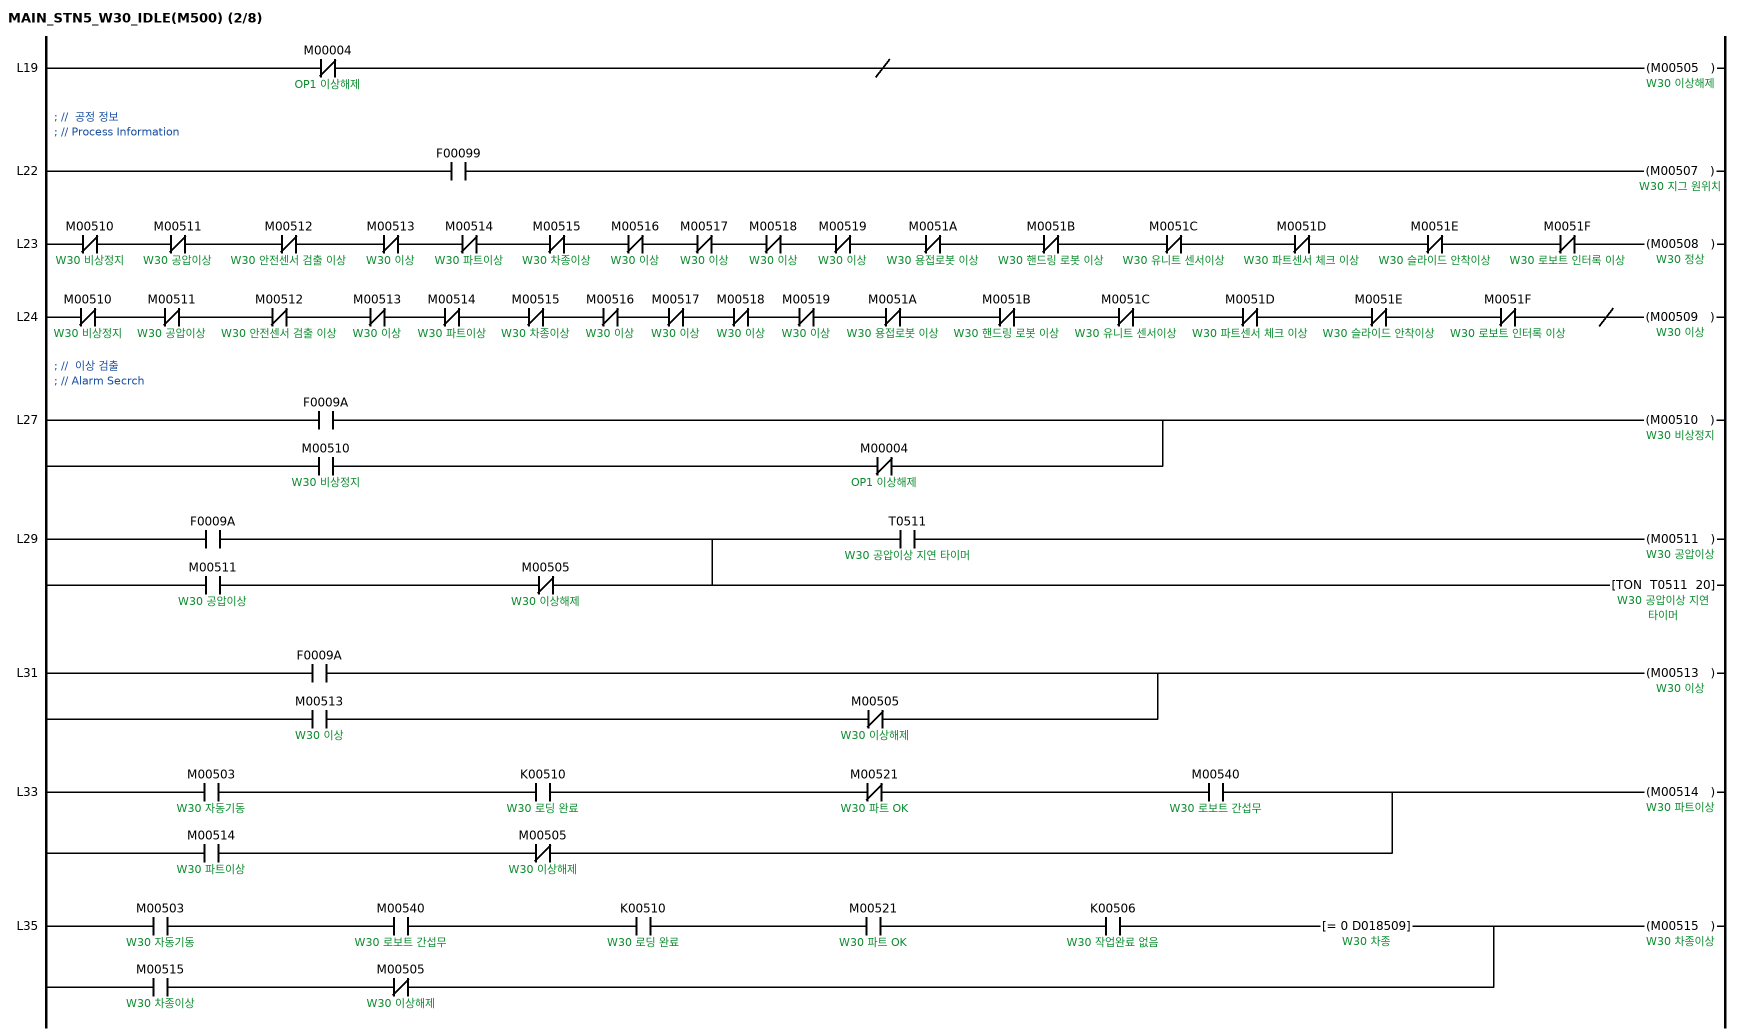
; L19
LOAD NOT  M00004	// OP1 이상해제
NOT
OUT       M00505	// W30 이상해제
//   //  공정 정보
//   // Process Information
; L22
LOAD      F00099
OUT       M00507	// W30 지그 원위치
; L23
LOAD NOT  M00510	// W30 비상정지
AND NOT   M00511	// W30 공압이상
AND NOT   M00512	// W30 안전센서 검출 이상
AND NOT   M00513	// W30 이상
AND NOT   M00514	// W30 파트이상
AND NOT   M00515	// W30 차종이상
AND NOT   M00516	// W30 이상
AND NOT   M00517	// W30 이상
AND NOT   M00518	// W30 이상
AND NOT   M00519	// W30 이상
AND NOT   M0051A	// W30 용접로봇 이상
AND NOT   M0051B	// W30 핸드링 로봇 이상
AND NOT   M0051C	// W30 유니트 센서이상
AND NOT   M0051D	// W30 파트센서 체크 이상
AND NOT   M0051E	// W30 슬라이드 안착이상
AND NOT   M0051F	// W30 로보트 인터록 이상
OUT       M00508	// W30 정상
; L24
LOAD NOT  M00510	// W30 비상정지
AND NOT   M00511	// W30 공압이상
AND NOT   M00512	// W30 안전센서 검출 이상
AND NOT   M00513	// W30 이상
AND NOT   M00514	// W30 파트이상
AND NOT   M00515	// W30 차종이상
AND NOT   M00516	// W30 이상
AND NOT   M00517	// W30 이상
AND NOT   M00518	// W30 이상
AND NOT   M00519	// W30 이상
AND NOT   M0051A	// W30 용접로봇 이상
AND NOT   M0051B	// W30 핸드링 로봇 이상
AND NOT   M0051C	// W30 유니트 센서이상
AND NOT   M0051D	// W30 파트센서 체크 이상
AND NOT   M0051E	// W30 슬라이드 안착이상
AND NOT   M0051F	// W30 로보트 인터록 이상
NOT
OUT       M00509	// W30 이상
//   //  이상 검출
//   // Alarm Secrch
; L27
LOAD      F0009A
LOAD      M00510	// W30 비상정지
AND NOT   M00004	// OP1 이상해제
OR LOAD
OUT       M00510	// W30 비상정지
; L29
LOAD      F0009A
LOAD      M00511	// W30 공압이상
AND NOT   M00505	// W30 이상해제
OR LOAD
MPUSH
AND       T0511	// W30 공압이상 지연 타이머
OUT       M00511	// W30 공압이상
MPOP
TON       T0511 20	// W30 공압이상 지연 타이머
; L31
LOAD      F0009A
LOAD      M00513	// W30 이상
AND NOT   M00505	// W30 이상해제
OR LOAD
OUT       M00513	// W30 이상
; L33
LOAD      M00503	// W30 자동기동
AND       K00510	// W30 로딩 완료
AND NOT   M00521	// W30 파트 OK
AND       M00540	// W30 로보트 간섭무
LOAD      M00514	// W30 파트이상
AND NOT   M00505	// W30 이상해제
OR LOAD
OUT       M00514	// W30 파트이상
; L35
LOAD      M00503	// W30 자동기동
AND       M00540	// W30 로보트 간섭무
AND       K00510	// W30 로딩 완료
AND       M00521	// W30 파트 OK
AND       K00506	// W30 작업완료 없음
AND=      0 D018509	// W30 차종
LOAD      M00515	// W30 차종이상
AND NOT   M00505	// W30 이상해제
OR LOAD
OUT       M00515	// W30 차종이상

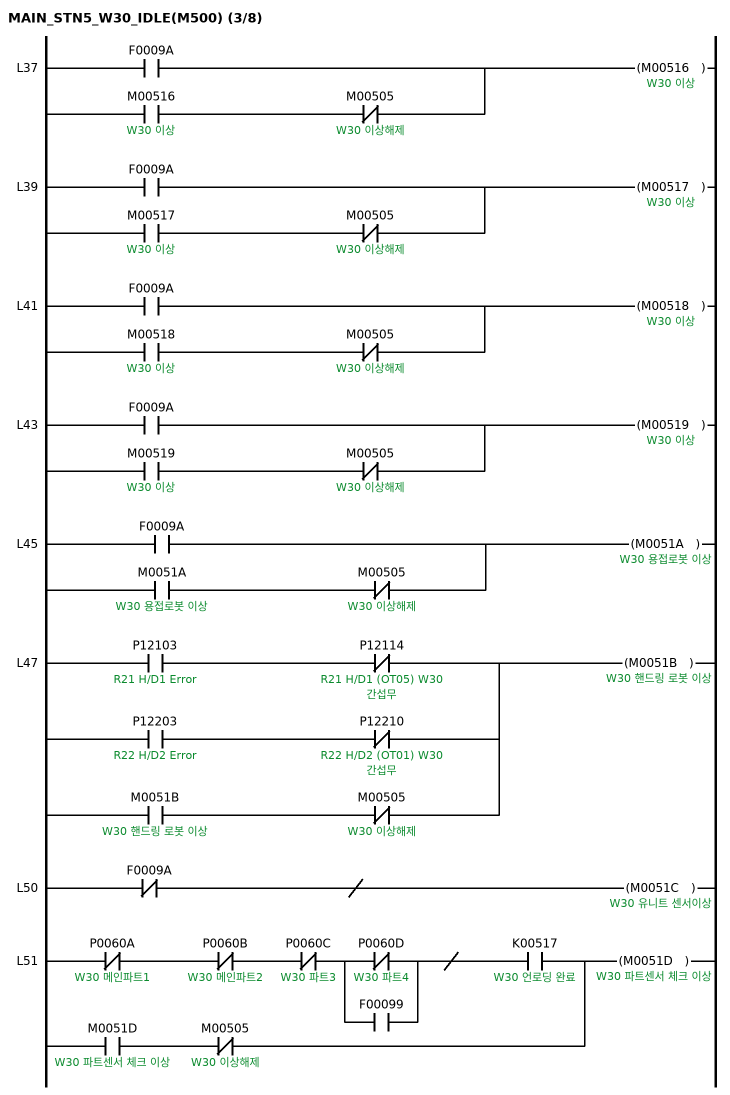
; L37
LOAD      F0009A
LOAD      M00516	// W30 이상
AND NOT   M00505	// W30 이상해제
OR LOAD
OUT       M00516	// W30 이상
; L39
LOAD      F0009A
LOAD      M00517	// W30 이상
AND NOT   M00505	// W30 이상해제
OR LOAD
OUT       M00517	// W30 이상
; L41
LOAD      F0009A
LOAD      M00518	// W30 이상
AND NOT   M00505	// W30 이상해제
OR LOAD
OUT       M00518	// W30 이상
; L43
LOAD      F0009A
LOAD      M00519	// W30 이상
AND NOT   M00505	// W30 이상해제
OR LOAD
OUT       M00519	// W30 이상
; L45
LOAD      F0009A
LOAD      M0051A	// W30 용접로봇 이상
AND NOT   M00505	// W30 이상해제
OR LOAD
OUT       M0051A	// W30 용접로봇 이상
; L47
LOAD      P12103	// R21 H/D1 Error
AND NOT   P12114	// R21 H/D1 (OT05) W30 간섭무
LOAD      P12203	// R22 H/D2 Error
AND NOT   P12210	// R22 H/D2 (OT01) W30 간섭무
OR LOAD
LOAD      M0051B	// W30 핸드링 로봇 이상
AND NOT   M00505	// W30 이상해제
OR LOAD
OUT       M0051B	// W30 핸드링 로봇 이상
; L50
LOAD NOT  F0009A
NOT
OUT       M0051C	// W30 유니트 센서이상
; L51
LOAD NOT  P0060A	// W30 메인파트1
AND NOT   P0060B	// W30 메인파트2
AND NOT   P0060C	// W30 파트3
LOAD NOT  P0060D	// W30 파트4
OR        F00099
AND LOAD
NOT
AND       K00517	// W30 언로딩 완료
LOAD      M0051D	// W30 파트센서 체크 이상
AND NOT   M00505	// W30 이상해제
OR LOAD
OUT       M0051D	// W30 파트센서 체크 이상

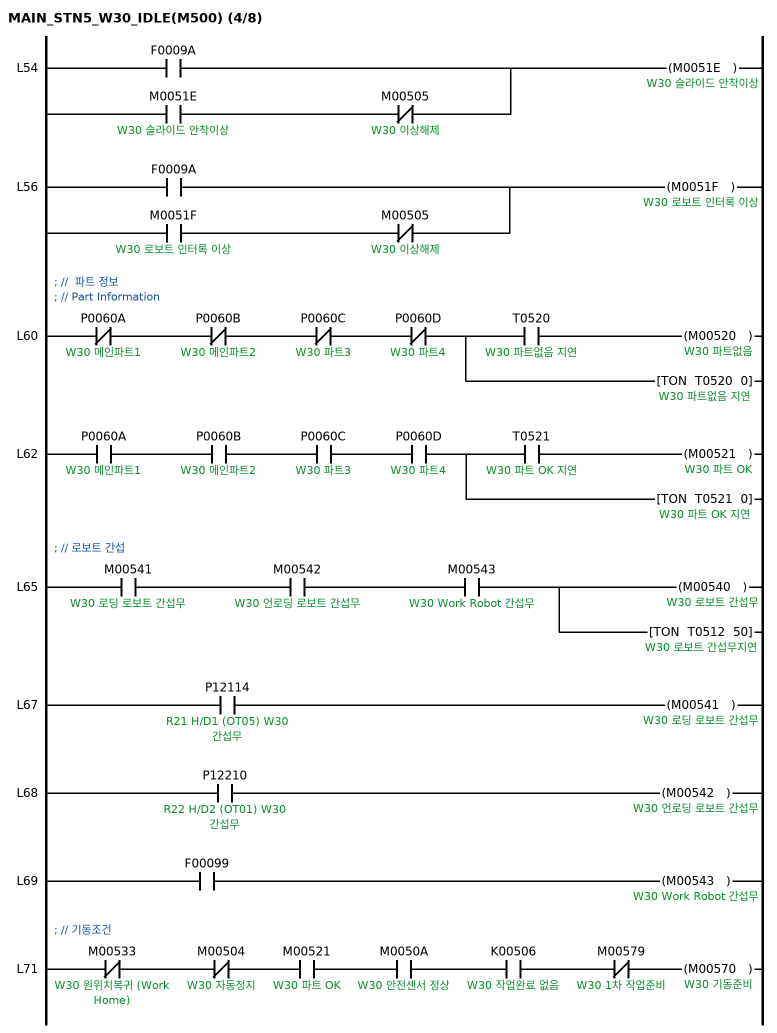
; L54
LOAD      F0009A
LOAD      M0051E	// W30 슬라이드 안착이상
AND NOT   M00505	// W30 이상해제
OR LOAD
OUT       M0051E	// W30 슬라이드 안착이상
; L56
LOAD      F0009A
LOAD      M0051F	// W30 로보트 인터록 이상
AND NOT   M00505	// W30 이상해제
OR LOAD
OUT       M0051F	// W30 로보트 인터록 이상
//   //  파트 정보
//   // Part Information
; L60
LOAD NOT  P0060A	// W30 메인파트1
AND NOT   P0060B	// W30 메인파트2
AND NOT   P0060C	// W30 파트3
AND NOT   P0060D	// W30 파트4
MPUSH
AND       T0520	// W30 파트없음 지연
OUT       M00520	// W30 파트없음
MPOP
TON       T0520 0	// W30 파트없음 지연
; L62
LOAD      P0060A	// W30 메인파트1
AND       P0060B	// W30 메인파트2
AND       P0060C	// W30 파트3
AND       P0060D	// W30 파트4
MPUSH
AND       T0521	// W30 파트 OK 지연
OUT       M00521	// W30 파트 OK
MPOP
TON       T0521 0	// W30 파트 OK 지연
//   // 로보트 간섭
; L65
LOAD      M00541	// W30 로딩 로보트 간섭무
AND       M00542	// W30 언로딩 로보트 간섭무
AND       M00543	// W30 Work Robot 간섭무
OUT       M00540	// W30 로보트 간섭무
TON       T0512 50	// W30 로보트 간섭무지연
; L67
LOAD      P12114	// R21 H/D1 (OT05) W30 간섭무
OUT       M00541	// W30 로딩 로보트 간섭무
; L68
LOAD      P12210	// R22 H/D2 (OT01) W30 간섭무
OUT       M00542	// W30 언로딩 로보트 간섭무
; L69
LOAD      F00099
OUT       M00543	// W30 Work Robot 간섭무
//   // 기동조건
; L71
LOAD NOT  M00533	// W30 원위치복귀 (Work Home)
AND NOT   M00504	// W30 자동정지
AND       M00521	// W30 파트 OK
AND       M0050A	// W30 안전센서 정상
AND       K00506	// W30 작업완료 없음
AND NOT   M00579	// W30 1차 작업준비
OUT       M00570	// W30 기동준비

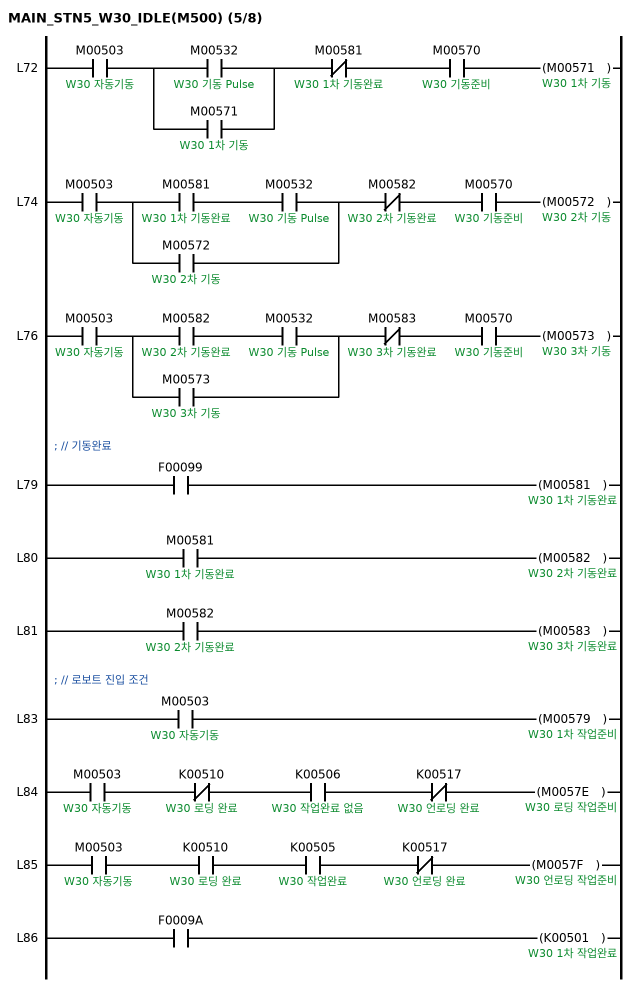
; L72
LOAD      M00503	// W30 자동기동
LOAD      M00532	// W30 기동 Pulse
OR        M00571	// W30 1차 기동
AND LOAD
AND NOT   M00581	// W30 1차 기동완료
AND       M00570	// W30 기동준비
OUT       M00571	// W30 1차 기동
; L74
LOAD      M00503	// W30 자동기동
LOAD      M00581	// W30 1차 기동완료
AND       M00532	// W30 기동 Pulse
OR        M00572	// W30 2차 기동
AND LOAD
AND NOT   M00582	// W30 2차 기동완료
AND       M00570	// W30 기동준비
OUT       M00572	// W30 2차 기동
; L76
LOAD      M00503	// W30 자동기동
LOAD      M00582	// W30 2차 기동완료
AND       M00532	// W30 기동 Pulse
OR        M00573	// W30 3차 기동
AND LOAD
AND NOT   M00583	// W30 3차 기동완료
AND       M00570	// W30 기동준비
OUT       M00573	// W30 3차 기동
//   // 기동완료
; L79
LOAD      F00099
OUT       M00581	// W30 1차 기동완료
; L80
LOAD      M00581	// W30 1차 기동완료
OUT       M00582	// W30 2차 기동완료
; L81
LOAD      M00582	// W30 2차 기동완료
OUT       M00583	// W30 3차 기동완료
//   // 로보트 진입 조건
; L83
LOAD      M00503	// W30 자동기동
OUT       M00579	// W30 1차 작업준비
; L84
LOAD      M00503	// W30 자동기동
AND NOT   K00510	// W30 로딩 완료
AND       K00506	// W30 작업완료 없음
AND NOT   K00517	// W30 언로딩 완료
OUT       M0057E	// W30 로딩 작업준비
; L85
LOAD      M00503	// W30 자동기동
AND       K00510	// W30 로딩 완료
AND       K00505	// W30 작업완료
AND NOT   K00517	// W30 언로딩 완료
OUT       M0057F	// W30 언로딩 작업준비
; L86
LOAD      F0009A
OUT       K00501	// W30 1차 작업완료

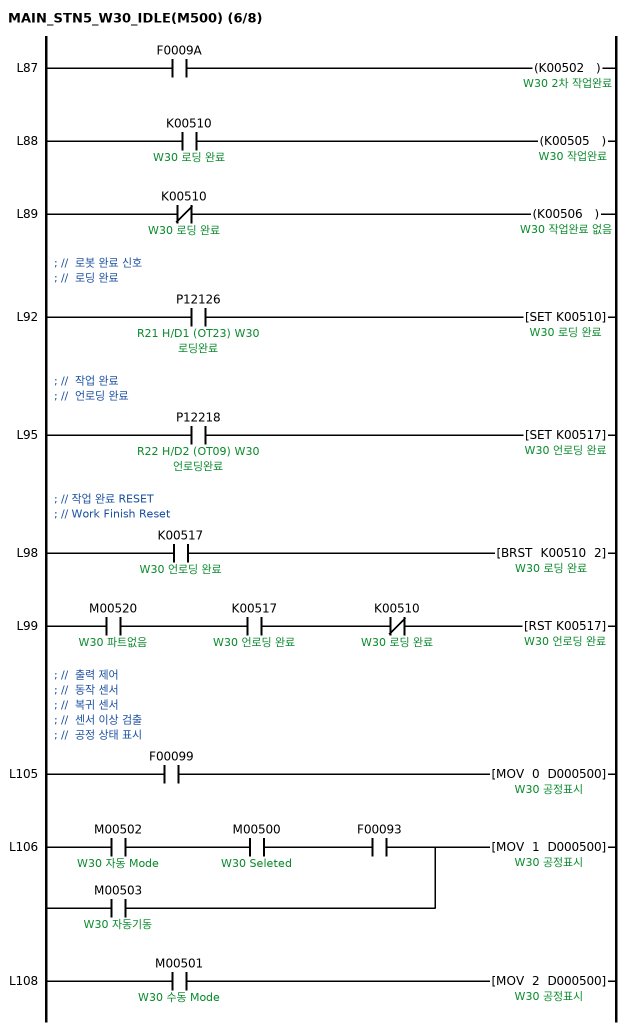
; L87
LOAD      F0009A
OUT       K00502	// W30 2차 작업완료
; L88
LOAD      K00510	// W30 로딩 완료
OUT       K00505	// W30 작업완료
; L89
LOAD NOT  K00510	// W30 로딩 완료
OUT       K00506	// W30 작업완료 없음
//   //  로봇 완료 신호
//   //  로딩 완료
; L92
LOAD      P12126	// R21 H/D1 (OT23) W30 로딩완료
SET       K00510	// W30 로딩 완료
//   //  작업 완료
//   //  언로딩 완료
; L95
LOAD      P12218	// R22 H/D2 (OT09) W30 언로딩완료
SET       K00517	// W30 언로딩 완료
//     // 작업 완료 RESET
//   // Work Finish Reset
; L98
LOAD      K00517	// W30 언로딩 완료
BRST      K00510 2	// W30 로딩 완료
; L99
LOAD      M00520	// W30 파트없음
AND       K00517	// W30 언로딩 완료
AND NOT   K00510	// W30 로딩 완료
RST       K00517	// W30 언로딩 완료
//     //  출력 제어
//   //  동작 센서
//   //  복귀 센서
//     //  센서 이상 검출
//   //  공정 상태 표시
; L105
LOAD      F00099
MOV       0 D000500	// W30 공정표시
; L106
LOAD      M00502	// W30 자동 Mode
AND       M00500	// W30 Seleted
AND       F00093
OR        M00503	// W30 자동기동
MOV       1 D000500	// W30 공정표시
; L108
LOAD      M00501	// W30 수동 Mode
MOV       2 D000500	// W30 공정표시

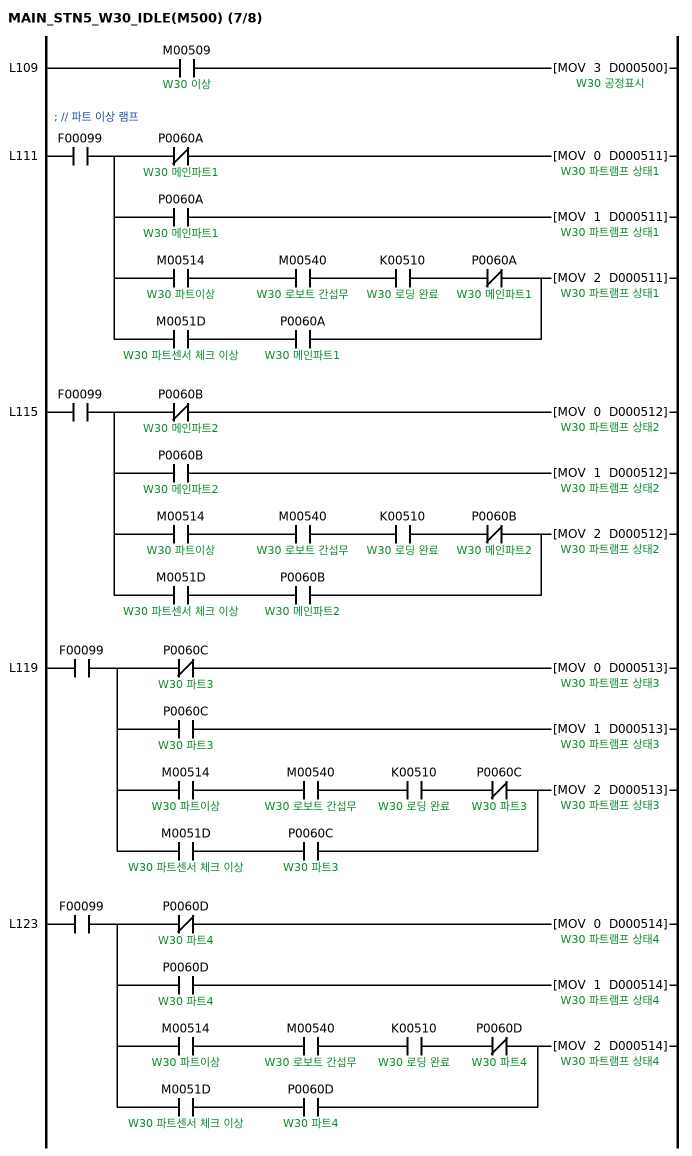
; L109
LOAD      M00509	// W30 이상
MOV       3 D000500	// W30 공정표시
//   // 파트 이상 램프
; L111
LOAD      F00099
MPUSH
AND NOT   P0060A	// W30 메인파트1
MOV       0 D000511	// W30 파트램프 상태1
MLOAD
AND       P0060A	// W30 메인파트1
MOV       1 D000511	// W30 파트램프 상태1
MPOP
LOAD      M00514	// W30 파트이상
AND       M00540	// W30 로보트 간섭무
AND       K00510	// W30 로딩 완료
AND NOT   P0060A	// W30 메인파트1
LOAD      M0051D	// W30 파트센서 체크 이상
AND       P0060A	// W30 메인파트1
OR LOAD
AND LOAD
MOV       2 D000511	// W30 파트램프 상태1
; L115
LOAD      F00099
MPUSH
AND NOT   P0060B	// W30 메인파트2
MOV       0 D000512	// W30 파트램프 상태2
MLOAD
AND       P0060B	// W30 메인파트2
MOV       1 D000512	// W30 파트램프 상태2
MPOP
LOAD      M00514	// W30 파트이상
AND       M00540	// W30 로보트 간섭무
AND       K00510	// W30 로딩 완료
AND NOT   P0060B	// W30 메인파트2
LOAD      M0051D	// W30 파트센서 체크 이상
AND       P0060B	// W30 메인파트2
OR LOAD
AND LOAD
MOV       2 D000512	// W30 파트램프 상태2
; L119
LOAD      F00099
MPUSH
AND NOT   P0060C	// W30 파트3
MOV       0 D000513	// W30 파트램프 상태3
MLOAD
AND       P0060C	// W30 파트3
MOV       1 D000513	// W30 파트램프 상태3
MPOP
LOAD      M00514	// W30 파트이상
AND       M00540	// W30 로보트 간섭무
AND       K00510	// W30 로딩 완료
AND NOT   P0060C	// W30 파트3
LOAD      M0051D	// W30 파트센서 체크 이상
AND       P0060C	// W30 파트3
OR LOAD
AND LOAD
MOV       2 D000513	// W30 파트램프 상태3
; L123
LOAD      F00099
MPUSH
AND NOT   P0060D	// W30 파트4
MOV       0 D000514	// W30 파트램프 상태4
MLOAD
AND       P0060D	// W30 파트4
MOV       1 D000514	// W30 파트램프 상태4
MPOP
LOAD      M00514	// W30 파트이상
AND       M00540	// W30 로보트 간섭무
AND       K00510	// W30 로딩 완료
AND NOT   P0060D	// W30 파트4
LOAD      M0051D	// W30 파트센서 체크 이상
AND       P0060D	// W30 파트4
OR LOAD
AND LOAD
MOV       2 D000514	// W30 파트램프 상태4

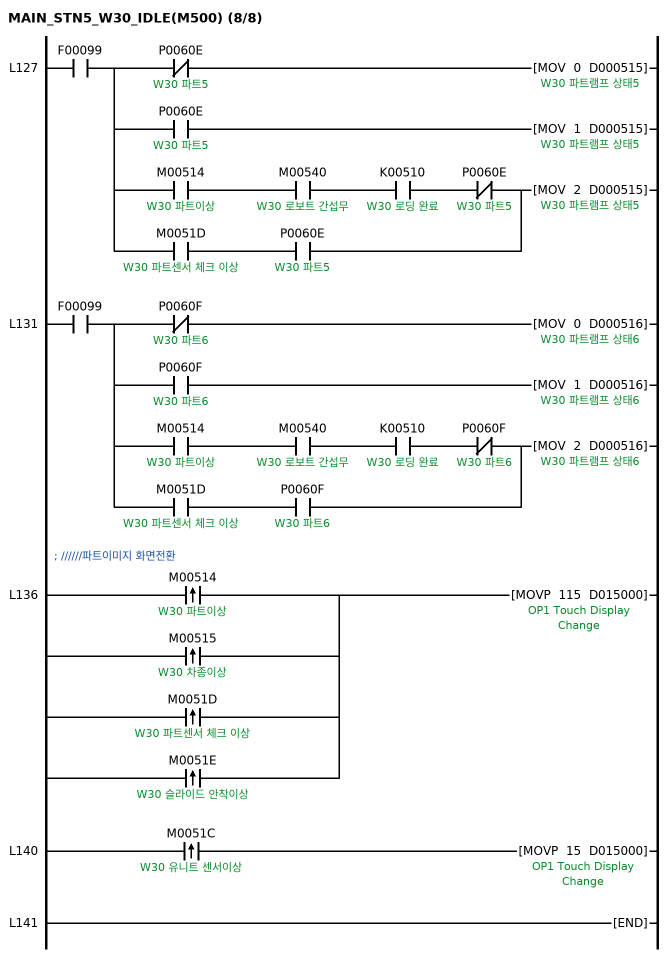
; L127
LOAD      F00099
MPUSH
AND NOT   P0060E	// W30 파트5
MOV       0 D000515	// W30 파트램프 상태5
MLOAD
AND       P0060E	// W30 파트5
MOV       1 D000515	// W30 파트램프 상태5
MPOP
LOAD      M00514	// W30 파트이상
AND       M00540	// W30 로보트 간섭무
AND       K00510	// W30 로딩 완료
AND NOT   P0060E	// W30 파트5
LOAD      M0051D	// W30 파트센서 체크 이상
AND       P0060E	// W30 파트5
OR LOAD
AND LOAD
MOV       2 D000515	// W30 파트램프 상태5
; L131
LOAD      F00099
MPUSH
AND NOT   P0060F	// W30 파트6
MOV       0 D000516	// W30 파트램프 상태6
MLOAD
AND       P0060F	// W30 파트6
MOV       1 D000516	// W30 파트램프 상태6
MPOP
LOAD      M00514	// W30 파트이상
AND       M00540	// W30 로보트 간섭무
AND       K00510	// W30 로딩 완료
AND NOT   P0060F	// W30 파트6
LOAD      M0051D	// W30 파트센서 체크 이상
AND       P0060F	// W30 파트6
OR LOAD
AND LOAD
MOV       2 D000516	// W30 파트램프 상태6
// //////파트이미지 화면전환
; L136
LOADP     M00514	// W30 파트이상
ORP       M00515	// W30 차종이상
ORP       M0051D	// W30 파트센서 체크 이상
ORP       M0051E	// W30 슬라이드 안착이상
MOVP      115 D015000	// OP1 Touch Display Change
; L140
LOADP     M0051C	// W30 유니트 센서이상
MOVP      15 D015000	// OP1 Touch Display Change
; L141
END

PROGRAM MAIN_STN6_W100(M700) (task: 스캔 프로그램)

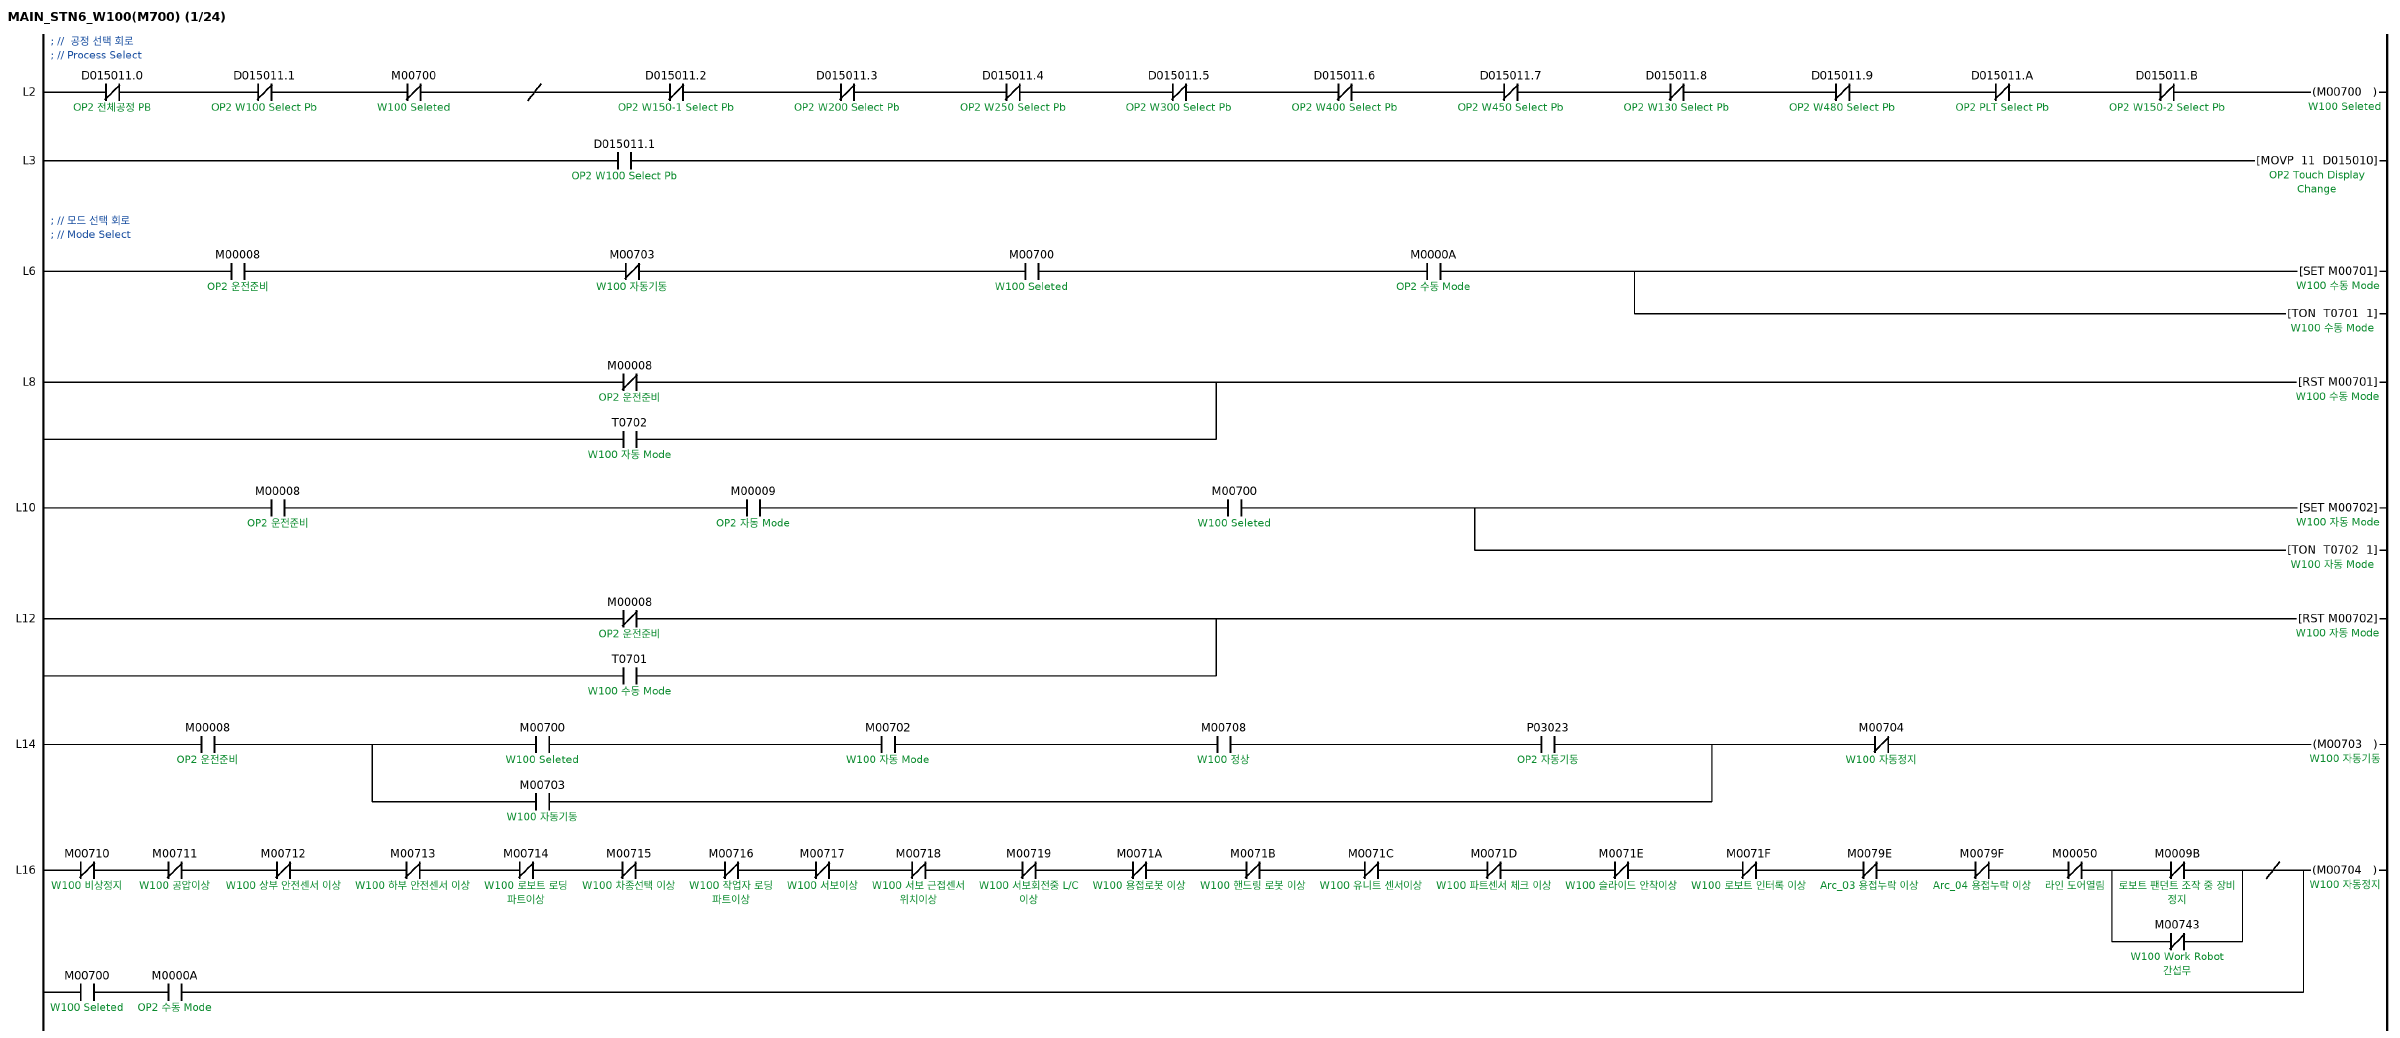
//   //  공정 선택 회로
//   // Process Select
; L2
LOAD NOT  D015011.0	// OP2 전체공정 PB
AND NOT   D015011.1	// OP2 W100 Select Pb
AND NOT   M00700	// W100 Seleted
NOT
AND NOT   D015011.2	// OP2 W150-1 Select Pb
AND NOT   D015011.3	// OP2 W200 Select Pb
AND NOT   D015011.4	// OP2 W250 Select Pb
AND NOT   D015011.5	// OP2 W300 Select Pb
AND NOT   D015011.6	// OP2 W400 Select Pb
AND NOT   D015011.7	// OP2 W450 Select Pb
AND NOT   D015011.8	// OP2 W130 Select Pb
AND NOT   D015011.9	// OP2 W480 Select Pb
AND NOT   D015011.A	// OP2 PLT Select Pb
AND NOT   D015011.B	// OP2 W150-2 Select Pb
OUT       M00700	// W100 Seleted
; L3
LOAD      D015011.1	// OP2 W100 Select Pb
MOVP      11 D015010	// OP2 Touch Display Change
// // 모드 선택 회로
//   // Mode Select
; L6
LOAD      M00008	// OP2 운전준비
AND NOT   M00703	// W100 자동기동
AND       M00700	// W100 Seleted
AND       M0000A	// OP2 수동 Mode
SET       M00701	// W100 수동 Mode
TON       T0701 1	// W100 수동 Mode
; L8
LOAD NOT  M00008	// OP2 운전준비
OR        T0702	// W100 자동 Mode
RST       M00701	// W100 수동 Mode
; L10
LOAD      M00008	// OP2 운전준비
AND       M00009	// OP2 자동 Mode
AND       M00700	// W100 Seleted
SET       M00702	// W100 자동 Mode
TON       T0702 1	// W100 자동 Mode
; L12
LOAD NOT  M00008	// OP2 운전준비
OR        T0701	// W100 수동 Mode
RST       M00702	// W100 자동 Mode
; L14
LOAD      M00008	// OP2 운전준비
LOAD      M00700	// W100 Seleted
AND       M00702	// W100 자동 Mode
AND       M00708	// W100 정상
AND       P03023	// OP2 자동기동
OR        M00703	// W100 자동기동
AND LOAD
AND NOT   M00704	// W100 자동정지
OUT       M00703	// W100 자동기동
; L16
LOAD NOT  M00710	// W100 비상정지
AND NOT   M00711	// W100 공압이상
AND NOT   M00712	// W100 상부 안전센서 이상
AND NOT   M00713	// W100 하부 안전센서 이상
AND NOT   M00714	// W100 로보트 로딩 파트이상
AND NOT   M00715	// W100 차종선택 이상
AND NOT   M00716	// W100 작업자 로딩 파트이상
AND NOT   M00717	// W100 서보이상
AND NOT   M00718	// W100 서보 근접센서 위치이상
AND NOT   M00719	// W100 서보회전중 L/C 이상
AND NOT   M0071A	// W100 용접로봇 이상
AND NOT   M0071B	// W100 핸드링 로봇 이상
AND NOT   M0071C	// W100 유니트 센서이상
AND NOT   M0071D	// W100 파트센서 체크 이상
AND NOT   M0071E	// W100 슬라이드 안착이상
AND NOT   M0071F	// W100 로보트 인터록 이상
AND NOT   M0079E	// Arc_03 용접누락 이상
AND NOT   M0079F	// Arc_04 용접누락 이상
AND NOT   M00050	// 라인 도어열림
LOAD NOT  M0009B	// 로보트 팬던트 조작 중 장비 정지
OR NOT    M00743	// W100 Work Robot 간섭무
AND LOAD
NOT
LOAD      M00700	// W100 Seleted
AND       M0000A	// OP2 수동 Mode
OR LOAD
OUT       M00704	// W100 자동정지

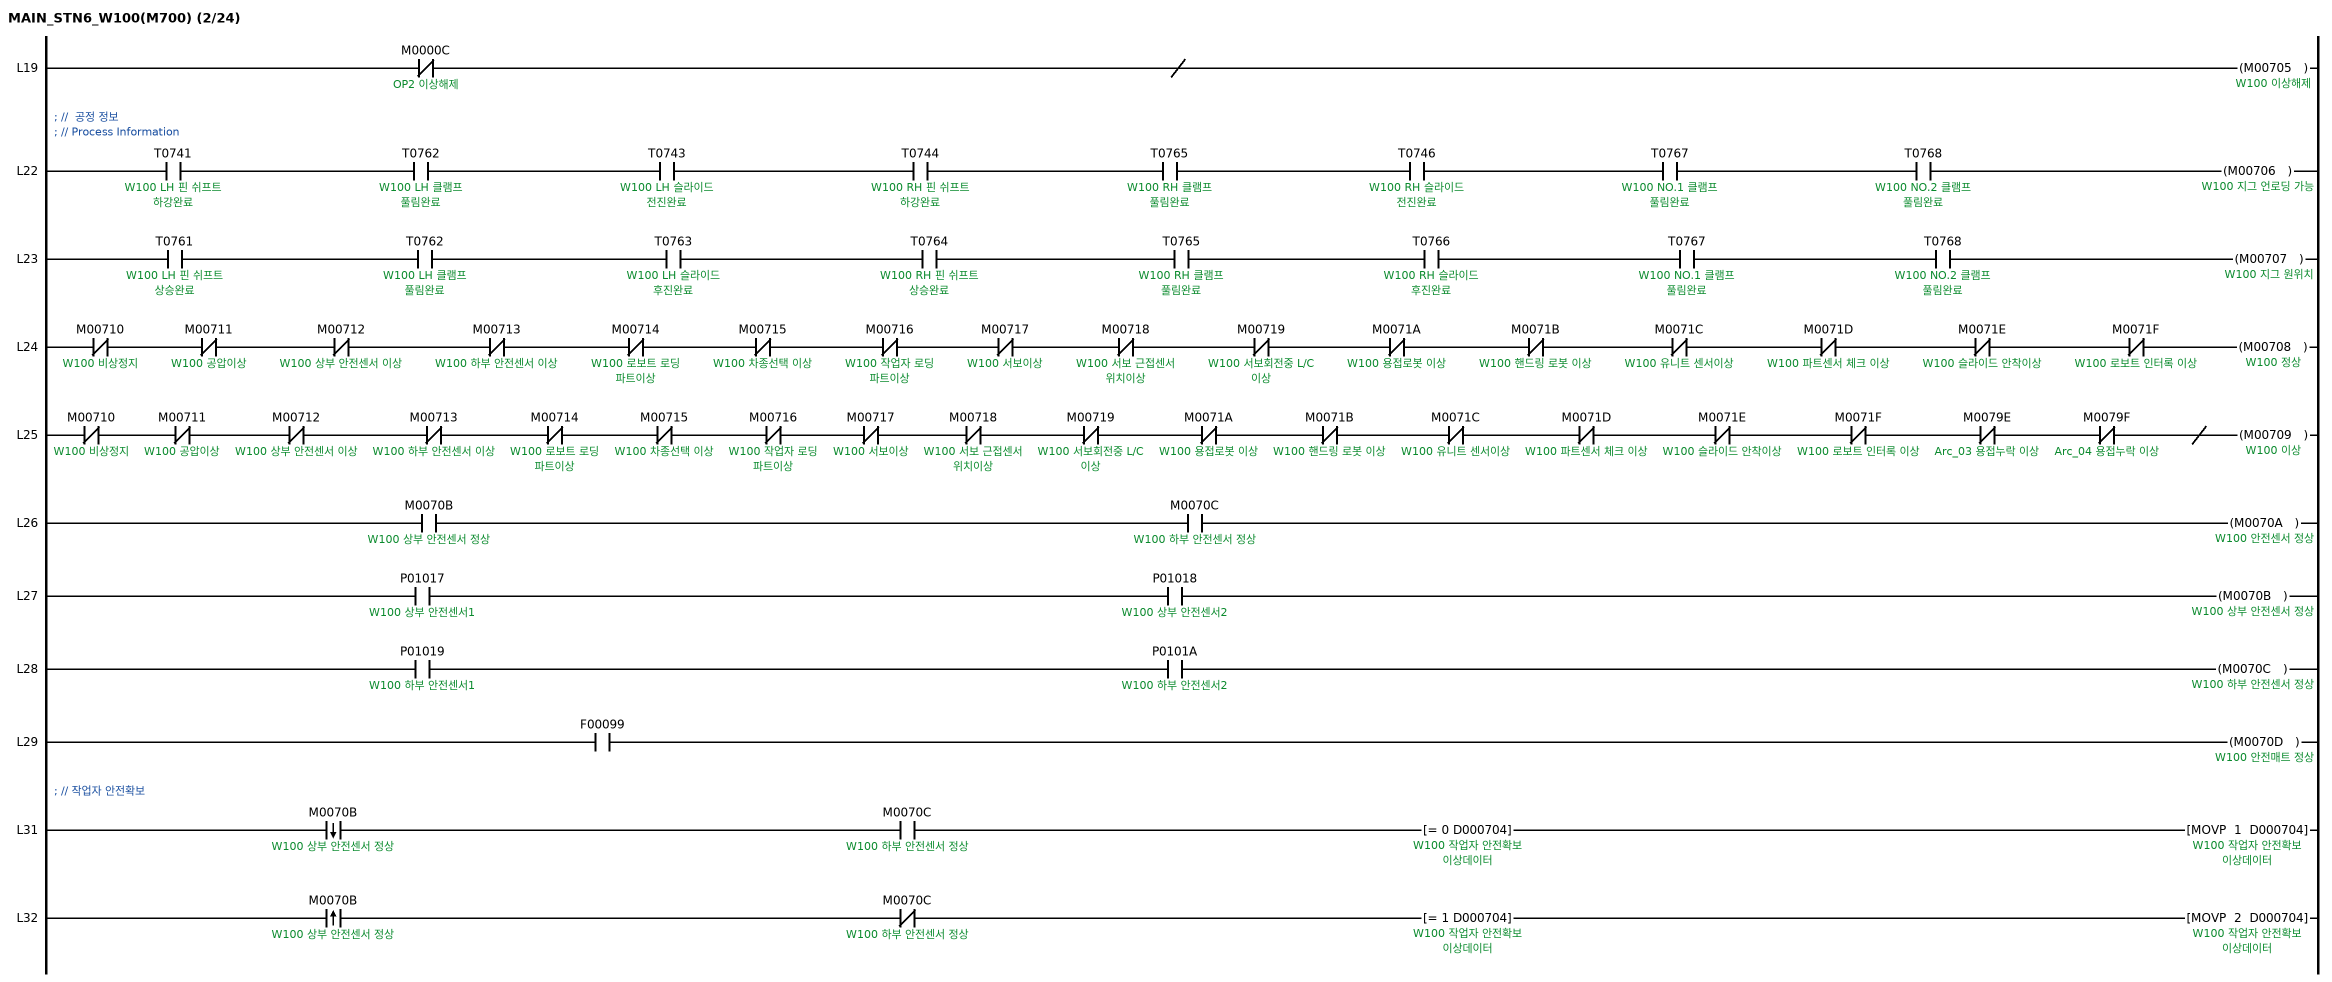
; L19
LOAD NOT  M0000C	// OP2 이상해제
NOT
OUT       M00705	// W100 이상해제
//   //  공정 정보
//   // Process Information
; L22
LOAD      T0741	// W100 LH 핀 쉬프트 하강완료
AND       T0762	// W100 LH 클램프 풀림완료
AND       T0743	// W100 LH 슬라이드 전진완료
AND       T0744	// W100 RH 핀 쉬프트 하강완료
AND       T0765	// W100 RH 클램프 풀림완료
AND       T0746	// W100 RH 슬라이드 전진완료
AND       T0767	// W100 NO.1 클램프 풀림완료
AND       T0768	// W100 NO.2 클램프 풀림완료
OUT       M00706	// W100 지그 언로딩 가능
; L23
LOAD      T0761	// W100 LH 핀 쉬프트 상승완료
AND       T0762	// W100 LH 클램프 풀림완료
AND       T0763	// W100 LH 슬라이드 후진완료
AND       T0764	// W100 RH 핀 쉬프트 상승완료
AND       T0765	// W100 RH 클램프 풀림완료
AND       T0766	// W100 RH 슬라이드 후진완료
AND       T0767	// W100 NO.1 클램프 풀림완료
AND       T0768	// W100 NO.2 클램프 풀림완료
OUT       M00707	// W100 지그 원위치
; L24
LOAD NOT  M00710	// W100 비상정지
AND NOT   M00711	// W100 공압이상
AND NOT   M00712	// W100 상부 안전센서 이상
AND NOT   M00713	// W100 하부 안전센서 이상
AND NOT   M00714	// W100 로보트 로딩 파트이상
AND NOT   M00715	// W100 차종선택 이상
AND NOT   M00716	// W100 작업자 로딩 파트이상
AND NOT   M00717	// W100 서보이상
AND NOT   M00718	// W100 서보 근접센서 위치이상
AND NOT   M00719	// W100 서보회전중 L/C 이상
AND NOT   M0071A	// W100 용접로봇 이상
AND NOT   M0071B	// W100 핸드링 로봇 이상
AND NOT   M0071C	// W100 유니트 센서이상
AND NOT   M0071D	// W100 파트센서 체크 이상
AND NOT   M0071E	// W100 슬라이드 안착이상
AND NOT   M0071F	// W100 로보트 인터록 이상
OUT       M00708	// W100 정상
; L25
LOAD NOT  M00710	// W100 비상정지
AND NOT   M00711	// W100 공압이상
AND NOT   M00712	// W100 상부 안전센서 이상
AND NOT   M00713	// W100 하부 안전센서 이상
AND NOT   M00714	// W100 로보트 로딩 파트이상
AND NOT   M00715	// W100 차종선택 이상
AND NOT   M00716	// W100 작업자 로딩 파트이상
AND NOT   M00717	// W100 서보이상
AND NOT   M00718	// W100 서보 근접센서 위치이상
AND NOT   M00719	// W100 서보회전중 L/C 이상
AND NOT   M0071A	// W100 용접로봇 이상
AND NOT   M0071B	// W100 핸드링 로봇 이상
AND NOT   M0071C	// W100 유니트 센서이상
AND NOT   M0071D	// W100 파트센서 체크 이상
AND NOT   M0071E	// W100 슬라이드 안착이상
AND NOT   M0071F	// W100 로보트 인터록 이상
AND NOT   M0079E	// Arc_03 용접누락 이상
AND NOT   M0079F	// Arc_04 용접누락 이상
NOT
OUT       M00709	// W100 이상
; L26
LOAD      M0070B	// W100 상부 안전센서 정상
AND       M0070C	// W100 하부 안전센서 정상
OUT       M0070A	// W100 안전센서 정상
; L27
LOAD      P01017	// W100 상부 안전센서1
AND       P01018	// W100 상부 안전센서2
OUT       M0070B	// W100 상부 안전센서 정상
; L28
LOAD      P01019	// W100 하부 안전센서1
AND       P0101A	// W100 하부 안전센서2
OUT       M0070C	// W100 하부 안전센서 정상
; L29
LOAD      F00099
OUT       M0070D	// W100 안전매트 정상
//    // 작업자 안전확보
; L31
LOADN     M0070B	// W100 상부 안전센서 정상
AND       M0070C	// W100 하부 안전센서 정상
AND=      0 D000704	// W100 작업자 안전확보 이상데이터
MOVP      1 D000704	// W100 작업자 안전확보 이상데이터
; L32
LOADP     M0070B	// W100 상부 안전센서 정상
AND NOT   M0070C	// W100 하부 안전센서 정상
AND=      1 D000704	// W100 작업자 안전확보 이상데이터
MOVP      2 D000704	// W100 작업자 안전확보 이상데이터

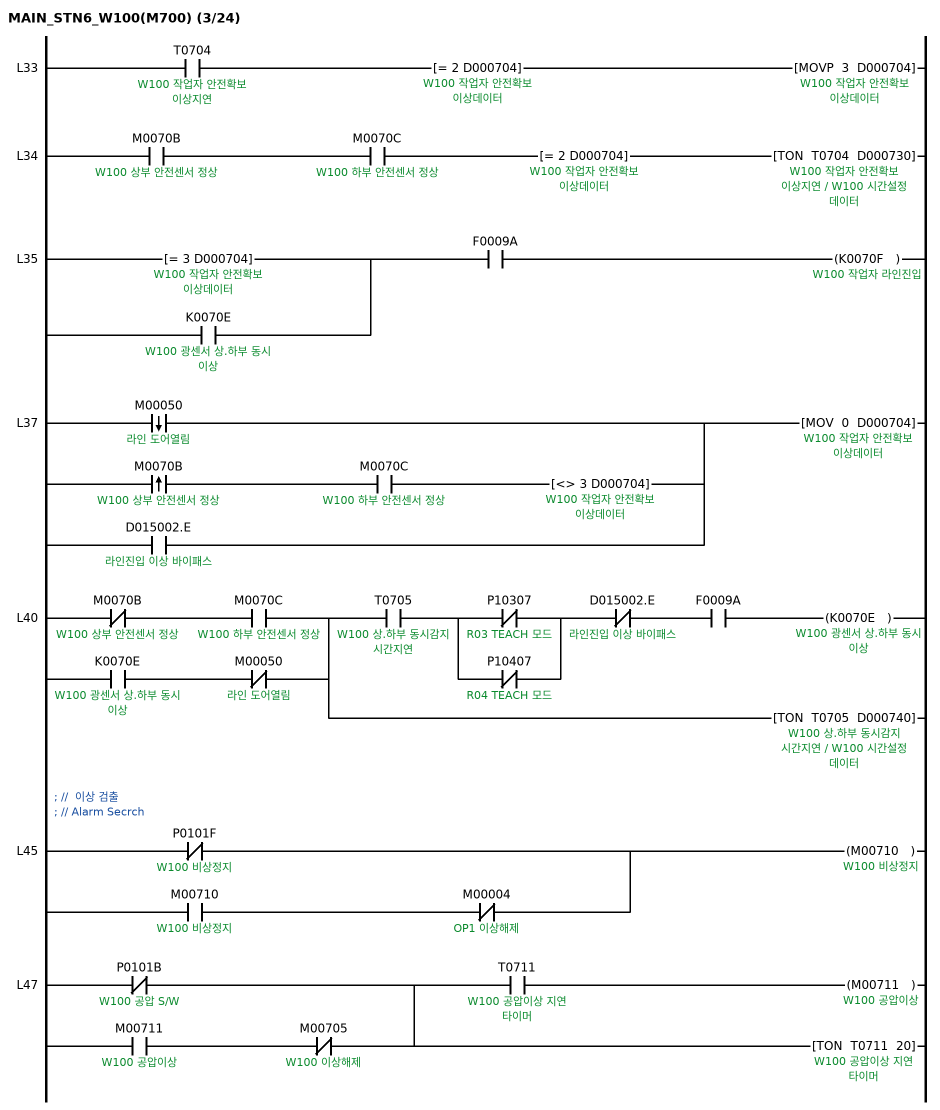
; L33
LOAD      T0704	// W100 작업자 안전확보 이상지연
AND=      2 D000704	// W100 작업자 안전확보 이상데이터
MOVP      3 D000704	// W100 작업자 안전확보 이상데이터
; L34
LOAD      M0070B	// W100 상부 안전센서 정상
AND       M0070C	// W100 하부 안전센서 정상
AND=      2 D000704	// W100 작업자 안전확보 이상데이터
TON       T0704 D000730	// W100 작업자 안전확보 이상지연 / W100 시간설정 데이터
; L35
LOAD=     3 D000704	// W100 작업자 안전확보 이상데이터
OR        K0070E	// W100 광센서 상.하부 동시 이상
AND       F0009A
OUT       K0070F	// W100 작업자 라인진입
; L37
LOADN     M00050	// 라인 도어열림
LOADP     M0070B	// W100 상부 안전센서 정상
AND       M0070C	// W100 하부 안전센서 정상
AND<>     3 D000704	// W100 작업자 안전확보 이상데이터
OR LOAD
OR        D015002.E	// 라인진입 이상 바이패스
MOV       0 D000704	// W100 작업자 안전확보 이상데이터
; L40
LOAD NOT  M0070B	// W100 상부 안전센서 정상
AND       M0070C	// W100 하부 안전센서 정상
LOAD      K0070E	// W100 광센서 상.하부 동시 이상
AND NOT   M00050	// 라인 도어열림
OR LOAD
MPUSH
AND       T0705	// W100 상.하부 동시감지 시간지연
LOAD NOT  P10307	// R03 TEACH 모드
OR NOT    P10407	// R04 TEACH 모드
AND LOAD
AND NOT   D015002.E	// 라인진입 이상 바이패스
AND       F0009A
OUT       K0070E	// W100 광센서 상.하부 동시 이상
MPOP
TON       T0705 D000740	// W100 상.하부 동시감지 시간지연 / W100 시간설정 데이터
//   //  이상 검출
//   // Alarm Secrch
; L45
LOAD NOT  P0101F	// W100 비상정지
LOAD      M00710	// W100 비상정지
AND NOT   M00004	// OP1 이상해제
OR LOAD
OUT       M00710	// W100 비상정지
; L47
LOAD NOT  P0101B	// W100 공압 S/W
LOAD      M00711	// W100 공압이상
AND NOT   M00705	// W100 이상해제
OR LOAD
MPUSH
AND       T0711	// W100 공압이상 지연 타이머
OUT       M00711	// W100 공압이상
MPOP
TON       T0711 20	// W100 공압이상 지연 타이머

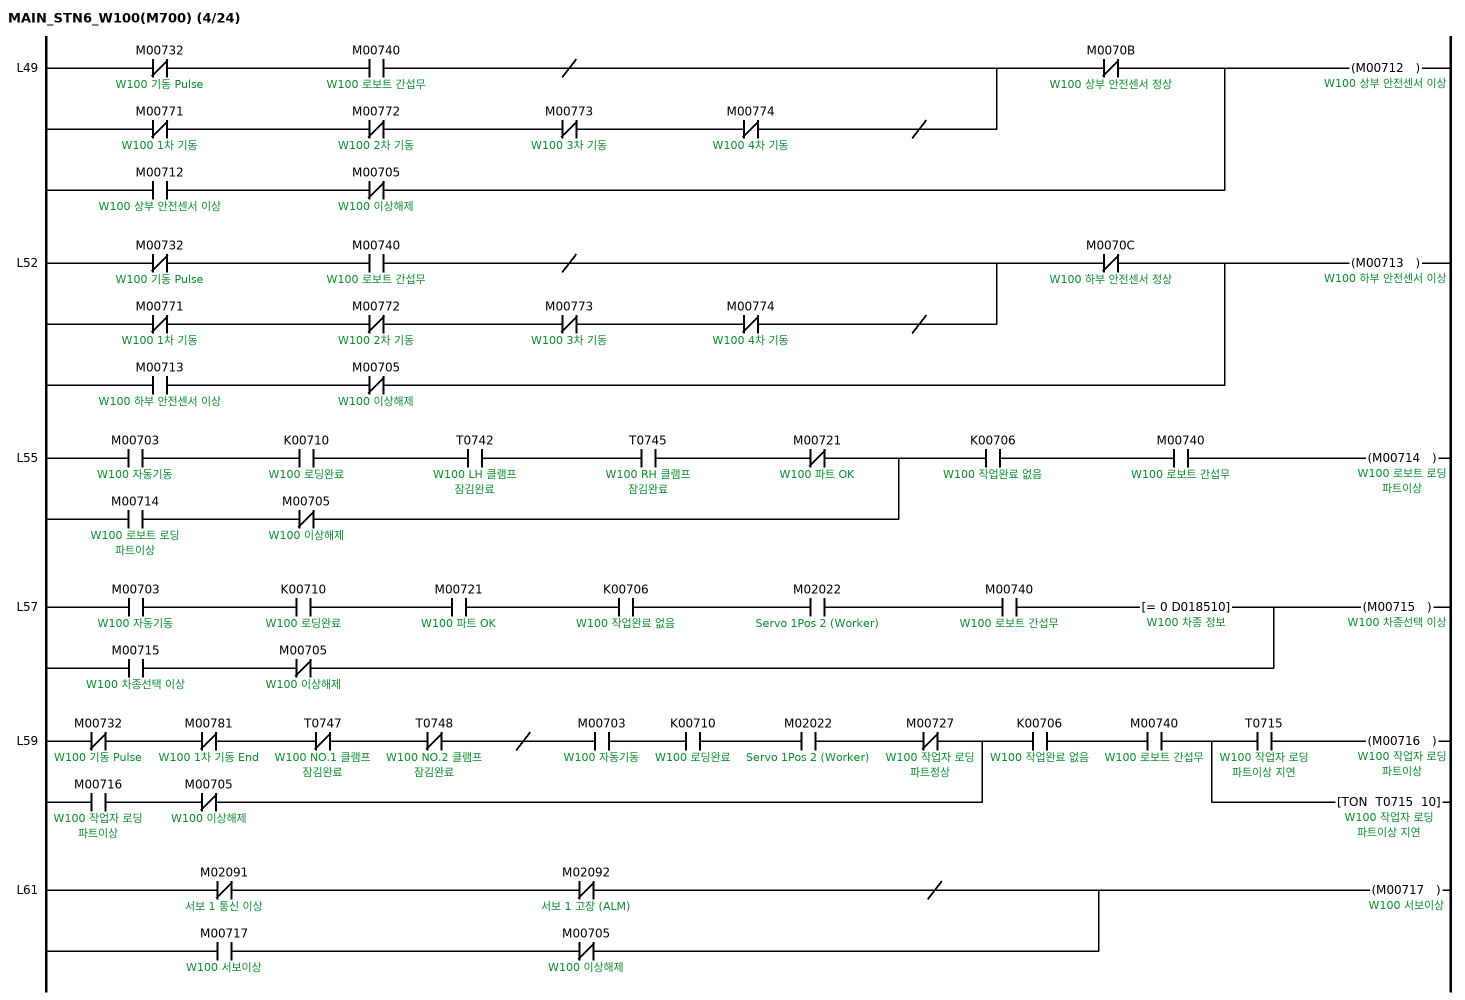
; L49
LOAD NOT  M00732	// W100 기동 Pulse
AND       M00740	// W100 로보트 간섭무
NOT
LOAD NOT  M00771	// W100 1차 기동
AND NOT   M00772	// W100 2차 기동
AND NOT   M00773	// W100 3차 기동
AND NOT   M00774	// W100 4차 기동
NOT
OR LOAD
AND NOT   M0070B	// W100 상부 안전센서 정상
LOAD      M00712	// W100 상부 안전센서 이상
AND NOT   M00705	// W100 이상해제
OR LOAD
OUT       M00712	// W100 상부 안전센서 이상
; L52
LOAD NOT  M00732	// W100 기동 Pulse
AND       M00740	// W100 로보트 간섭무
NOT
LOAD NOT  M00771	// W100 1차 기동
AND NOT   M00772	// W100 2차 기동
AND NOT   M00773	// W100 3차 기동
AND NOT   M00774	// W100 4차 기동
NOT
OR LOAD
AND NOT   M0070C	// W100 하부 안전센서 정상
LOAD      M00713	// W100 하부 안전센서 이상
AND NOT   M00705	// W100 이상해제
OR LOAD
OUT       M00713	// W100 하부 안전센서 이상
; L55
LOAD      M00703	// W100 자동기동
AND       K00710	// W100 로딩완료
AND       T0742	// W100 LH 클램프 잠김완료
AND       T0745	// W100 RH 클램프 잠김완료
AND NOT   M00721	// W100 파트 OK
LOAD      M00714	// W100 로보트 로딩 파트이상
AND NOT   M00705	// W100 이상해제
OR LOAD
AND       K00706	// W100 작업완료 없음
AND       M00740	// W100 로보트 간섭무
OUT       M00714	// W100 로보트 로딩 파트이상
; L57
LOAD      M00703	// W100 자동기동
AND       K00710	// W100 로딩완료
AND       M00721	// W100 파트 OK
AND       K00706	// W100 작업완료 없음
AND       M02022	// Servo 1Pos 2 (Worker)
AND       M00740	// W100 로보트 간섭무
AND=      0 D018510	// W100 차종 정보
LOAD      M00715	// W100 차종선택 이상
AND NOT   M00705	// W100 이상해제
OR LOAD
OUT       M00715	// W100 차종선택 이상
; L59
LOAD NOT  M00732	// W100 기동 Pulse
AND NOT   M00781	// W100 1차 기동 End
AND NOT   T0747	// W100 NO.1 클램프 잠김완료
AND NOT   T0748	// W100 NO.2 클램프 잠김완료
NOT
AND       M00703	// W100 자동기동
AND       K00710	// W100 로딩완료
AND       M02022	// Servo 1Pos 2 (Worker)
AND NOT   M00727	// W100 작업자 로딩 파트정상
LOAD      M00716	// W100 작업자 로딩 파트이상
AND NOT   M00705	// W100 이상해제
OR LOAD
AND       K00706	// W100 작업완료 없음
AND       M00740	// W100 로보트 간섭무
MPUSH
AND       T0715	// W100 작업자 로딩 파트이상 지연
OUT       M00716	// W100 작업자 로딩 파트이상
MPOP
TON       T0715 10	// W100 작업자 로딩 파트이상 지연
; L61
LOAD NOT  M02091	// 서보 1 통신 이상
AND NOT   M02092	// 서보 1 고장 (ALM)
NOT
LOAD      M00717	// W100 서보이상
AND NOT   M00705	// W100 이상해제
OR LOAD
OUT       M00717	// W100 서보이상

